C03637=1030.012,334.966,368.080,171.691,46.330,159.041
C03638=1030.005,334.718,368.116,171.685,46.330,159.040
C03639=1029.998,334.472,368.152,171.679,46.328,159.039
C03640=1029.990,334.224,368.188,171.674,46.328,159.038
C03641=1029.982,333.977,368.224,171.668,46.327,159.038
C03642=1029.975,333.730,368.260,171.662,46.326,159.037
C03643=1029.968,333.482,368.296,171.656,46.326,159.036
C03644=1029.961,333.235,368.331,171.652,46.326,159.035
C03645=1029.953,332.988,368.368,171.646,46.325,159.034
C03646=1029.945,332.740,368.403,171.640,46.325,159.034
C03647=1029.938,332.493,368.438,171.635,46.324,159.033
C03648=1029.930,332.246,368.475,171.629,46.323,159.032
C03649=1029.924,331.998,368.510,171.623,46.323,159.031
C03650=1029.916,331.751,368.546,171.617,46.322,159.030
C03651=1029.909,331.504,368.581,171.612,46.321,159.030
C03652=1029.901,331.256,368.617,171.606,46.321,159.029
C03653=1029.895,331.009,368.653,171.601,46.321,159.028
C03654=1029.886,330.762,368.688,171.596,46.320,159.027
C03655=1029.879,330.514,368.723,171.590,46.319,159.027
C03656=1029.872,330.267,368.759,171.584,46.319,159.026
C03657=1029.865,330.019,368.795,171.579,46.319,159.025
C03658=1029.857,329.772,368.831,171.574,46.318,159.024
C03659=1029.851,329.525,368.866,171.569,46.317,159.024
C03660=1029.843,329.277,368.902,171.563,46.317,159.023
C03661=1029.835,329.030,368.937,171.557,46.317,159.022
C03662=1029.829,328.783,368.972,171.552,46.316,159.021
C03663=1029.821,328.535,369.008,171.546,46.315,159.021
C03664=1029.814,328.288,369.043,171.541,46.316,159.020
C03665=1029.807,328.040,369.079,171.536,46.315,159.019
C03666=1029.800,327.793,369.115,171.530,46.314,159.018
C03667=1029.792,327.546,369.149,171.525,46.314,159.018
C03668=1029.785,327.298,369.185,171.519,46.313,159.017
C03669=1029.777,327.051,369.219,171.514,46.313,159.016
C03670=1029.769,326.803,369.254,171.509,46.313,159.015
C03671=1029.762,326.556,369.289,171.503,46.313,159.015
C03672=1029.755,326.309,369.324,171.498,46.313,159.014
C03673=1029.748,326.061,369.359,171.493,46.312,159.013
C03674=1029.740,325.814,369.394,171.487,46.312,159.013
C03675=1029.733,325.566,369.429,171.482,46.311,159.012
C03676=1029.725,325.319,369.464,171.477,46.311,159.011
C03677=1029.718,325.071,369.498,171.471,46.311,159.011
C03678=1029.711,324.824,369.533,171.466,46.310,159.010
C03679=1029.703,324.576,369.568,171.460,46.310,159.009
C03680=1029.696,324.329,369.604,171.456,46.310,159.009
C03681=1029.689,324.081,369.637,171.450,46.310,159.008
C03682=1029.682,323.833,369.673,171.444,46.310,159.007
C03683=1029.674,323.586,369.707,171.440,46.310,159.007
C03684=1029.666,323.339,369.742,171.434,46.310,159.006
C03685=1029.660,323.092,369.777,171.429,46.309,159.005
C03686=1029.652,322.844,369.812,171.424,46.309,159.005
C03687=1029.645,322.596,369.846,171.419,46.309,159.004
C03688=1029.638,322.349,369.881,171.413,46.309,159.003
C03689=1029.630,322.102,369.915,171.408,46.308,159.003
C03690=1029.624,321.891,369.946,171.404,46.308,159.002
C03691=1029.618,321.680,369.974,171.399,46.308,159.002
C03692=1029.612,321.470,370.004,171.395,46.308,159.001
C03693=1029.605,321.259,370.033,171.390,46.308,159.000
C03694=1029.600,321.049,370.063,171.386,46.307,159.000
C03695=1029.593,320.838,370.093,171.381,46.307,158.999
C03696=1029.588,320.627,370.122,171.377,46.307,158.999
C03697=1029.581,320.417,370.151,171.373,46.307,158.998
C03698=1029.575,320.169,370.186,171.367,46.307,158.998
C03699=1029.567,319.922,370.220,171.363,46.306,158.997
C03700=1029.560,319.674,370.255,171.357,46.306,158.996
C03701=1029.553,319.426,370.289,171.352,46.306,158.996
C03702=1029.545,319.179,370.324,171.347,46.306,158.995
C03703=1029.539,318.931,370.358,171.342,46.306,158.994
C03704=1029.531,318.684,370.393,171.337,46.306,158.994
C03705=1029.525,318.436,370.427,171.332,46.306,158.993
C03706=1029.517,318.189,370.462,171.327,46.306,158.993
C03707=1029.510,317.941,370.495,171.322,46.306,158.992
C03708=1029.503,317.694,370.531,171.317,46.305,158.991
C03709=1029.496,317.446,370.564,171.311,46.305,158.991
C03710=1029.489,317.199,370.599,171.307,46.305,158.990
C03711=1029.482,316.951,370.633,171.301,46.305,158.989
C03712=1029.475,316.703,370.667,171.297,46.305,158.989
C03713=1029.468,316.456,370.702,171.291,46.305,158.988
C03714=1029.462,316.209,370.736,171.286,46.305,158.988
C03715=1029.454,315.961,370.770,171.282,46.305,158.987
C03716=1029.448,315.714,370.805,171.276,46.305,158.987
C03717=1029.440,315.466,370.839,171.272,46.305,158.986
C03718=1029.433,315.219,370.872,171.266,46.305,158.985
C03719=1029.427,314.971,370.907,171.262,46.305,158.985
C03720=1029.419,314.724,370.941,171.257,46.305,158.984
C03721=1029.412,314.476,370.975,171.251,46.305,158.984
C03722=1029.406,314.229,371.009,171.247,46.305,158.983
C03723=1029.399,313.981,371.043,171.241,46.305,158.982
C03724=1029.392,313.734,371.078,171.237,46.305,158.982
C03725=1029.385,313.486,371.112,171.232,46.305,158.981
C03726=1029.378,313.238,371.146,171.227,46.305,158.981
C03727=1029.371,312.991,371.180,171.222,46.305,158.980
C03728=1029.365,312.743,371.214,171.218,46.305,158.980
C03729=1029.358,312.496,371.248,171.212,46.305,158.979
C03730=1029.351,312.248,371.282,171.207,46.305,158.978
C03731=1029.344,312.000,371.316,171.203,46.305,158.978
C03732=1029.337,311.753,371.349,171.197,46.305,158.977
C03733=1029.331,311.505,371.384,171.193,46.305,158.977
C03734=1029.324,311.257,371.417,171.188,46.305,158.976
C03735=1029.317,311.010,371.451,171.183,46.306,158.976
C03736=1029.310,310.763,371.485,171.178,46.305,158.975
C03737=1029.303,310.515,371.519,171.174,46.306,158.975
C03738=1029.295,310.268,371.552,171.168,46.306,158.974
C03739=1029.288,310.019,371.585,171.164,46.306,158.974
C03740=1029.281,309.772,371.618,171.158,46.306,158.973
C03741=1029.273,309.525,371.652,171.154,46.307,158.973
C03742=1029.266,309.277,371.685,171.149,46.306,158.972
C03743=1029.259,309.029,371.719,171.144,46.307,158.972
C03744=1029.253,308.782,371.752,171.140,46.307,158.971
C03745=1029.245,308.535,371.785,171.134,46.307,158.970
C03746=1029.238,308.286,371.818,171.130,46.308,158.970
C03747=1029.231,308.040,371.852,171.126,46.308,158.970
C03748=1029.224,307.791,371.885,171.120,46.308,158.969
C03749=1029.216,307.544,371.918,171.116,46.309,158.969
C03750=1029.205,307.127,371.974,171.108,46.309,158.968
C03751=1029.193,306.711,372.030,171.099,46.309,158.967
C03752=1029.181,306.295,372.086,171.091,46.310,158.966
C03753=1029.170,305.879,372.141,171.084,46.311,158.965
C03754=1029.162,305.631,372.175,171.079,46.311,158.965
C03755=1029.155,305.384,372.207,171.074,46.312,158.964
C03756=1029.148,305.136,372.241,171.069,46.311,158.964
C03757=1029.141,304.888,372.274,171.065,46.312,158.963
C03758=1029.134,304.640,372.306,171.060,46.312,158.963
C03759=1029.127,304.393,372.340,171.055,46.313,158.963
C03760=1029.121,304.145,372.373,171.051,46.313,158.962
C03761=1029.113,303.897,372.405,171.046,46.313,158.961
C03762=1029.107,303.650,372.439,171.041,46.314,158.961
C03763=1029.100,303.402,372.472,171.037,46.314,158.961
C03764=1029.093,303.154,372.505,171.033,46.314,158.960
C03765=1029.085,302.907,372.538,171.027,46.315,158.960
C03766=1029.079,302.659,372.571,171.023,46.316,158.959
C03767=1029.072,302.411,372.604,171.019,46.316,158.959
C03768=1029.065,302.164,372.636,171.014,46.316,158.958
C03769=1029.058,301.916,372.670,171.009,46.316,158.958
C03770=1029.052,301.668,372.702,171.004,46.317,158.957
C03771=1029.044,301.420,372.735,171.000,46.317,158.957
C03772=1029.038,301.173,372.768,170.996,46.318,158.957
C03773=1029.031,300.925,372.801,170.990,46.318,158.956
C03774=1029.025,300.677,372.834,170.986,46.319,158.956
C03775=1029.017,300.430,372.867,170.982,46.319,158.955
C03776=1029.010,300.182,372.900,170.977,46.319,158.955
C03777=1029.004,299.934,372.932,170.973,46.320,158.954
C03778=1028.996,299.686,372.965,170.968,46.320,158.954
C03779=1028.990,299.439,372.998,170.963,46.321,158.954
C03780=1028.983,299.191,373.031,170.959,46.321,158.953
C03781=1028.976,298.943,373.063,170.955,46.322,158.953
C03782=1028.970,298.696,373.096,170.950,46.322,158.952
C03783=1028.963,298.447,373.129,170.945,46.323,158.952
C03784=1028.956,298.200,373.161,170.941,46.323,158.951
C03785=1028.950,297.953,373.194,170.936,46.323,158.951
C03786=1028.943,297.704,373.227,170.932,46.324,158.951
C03787=1028.936,297.457,373.259,170.928,46.324,158.950
C03788=1028.930,297.209,373.292,170.922,46.325,158.950
C03789=1028.923,296.962,373.324,170.918,46.325,158.949
C03790=1028.916,296.714,373.357,170.914,46.326,158.949
C03791=1028.909,296.466,373.390,170.909,46.326,158.948
C03792=1028.903,296.219,373.422,170.905,46.327,158.948
C03793=1028.896,295.970,373.454,170.901,46.328,158.948
C03794=1028.889,295.722,373.487,170.897,46.328,158.947
C03795=1028.883,295.475,373.520,170.891,46.329,158.947
C03796=1028.876,295.228,373.552,170.887,46.329,158.946
C03797=1028.870,294.980,373.584,170.883,46.329,158.946
C03798=1028.863,294.732,373.618,170.878,46.330,158.946
C03799=1028.856,294.484,373.649,170.874,46.331,158.945
C03800=1028.850,294.236,373.682,170.870,46.331,158.945
C03801=1028.843,293.989,373.714,170.866,46.332,158.945
C03802=1028.836,293.740,373.746,170.860,46.332,158.944
C03803=1028.829,293.493,373.778,170.856,46.333,158.944
C03804=1028.822,293.245,373.811,170.852,46.334,158.943
C03805=1028.816,292.997,373.843,170.848,46.334,158.943
C03806=1028.804,292.598,373.894,170.840,46.335,158.942
C03807=1028.794,292.199,373.946,170.834,46.336,158.942
C03808=1028.783,291.800,373.998,170.827,46.337,158.941
C03809=1028.772,291.400,374.049,170.820,46.339,158.941
C03810=1028.765,291.153,374.081,170.815,46.339,158.940
C03811=1028.759,290.905,374.113,170.811,46.340,158.940
C03812=1028.752,290.657,374.145,170.807,46.341,158.940
C03813=1028.745,290.409,374.176,170.803,46.341,158.939
C03814=1028.738,290.161,374.208,170.799,46.342,158.939
C03815=1028.731,289.914,374.240,170.793,46.343,158.939
C03816=1028.725,289.665,374.272,170.789,46.344,158.938
C03817=1028.718,289.417,374.304,170.785,46.344,158.938
C03818=1028.711,289.170,374.336,170.781,46.345,158.938
C03819=1028.704,288.922,374.367,170.777,46.346,158.938
C03820=1028.697,288.674,374.399,170.772,46.347,158.937
C03821=1028.690,288.427,374.431,170.768,46.348,158.937
C03822=1028.684,288.179,374.463,170.764,46.348,158.936
C03823=1028.677,287.930,374.495,170.759,46.350,158.936
C03824=1028.670,287.682,374.526,170.755,46.350,158.936
C03825=1028.664,287.434,374.558,170.751,46.351,158.935
C03826=1028.657,287.187,374.590,170.747,46.352,158.935
C03827=1028.650,286.939,374.621,170.742,46.352,158.935
C03828=1028.643,286.691,374.653,170.738,46.353,158.935
C03829=1028.636,286.443,374.684,170.734,46.354,158.934
C03830=1028.630,286.196,374.716,170.730,46.355,158.934
C03831=1028.624,285.947,374.748,170.726,46.356,158.934
C03832=1028.617,285.699,374.779,170.722,46.357,158.933
C03833=1028.609,285.452,374.810,170.717,46.357,158.933
C03834=1028.603,285.204,374.841,170.712,46.359,158.933
C03835=1028.596,284.956,374.873,170.708,46.360,158.932
C03836=1028.589,284.708,374.904,170.704,46.361,158.932
C03837=1028.583,284.460,374.936,170.700,46.361,158.932
C03838=1028.576,284.212,374.967,170.696,46.362,158.932
C03839=1028.569,283.964,374.999,170.692,46.363,158.931
C03840=1028.562,283.716,375.030,170.688,46.364,158.931
C03841=1028.556,283.469,375.061,170.684,46.365,158.931
C03842=1028.548,283.221,375.092,170.680,46.366,158.931
C03843=1028.542,282.973,375.124,170.676,46.367,158.930
C03844=1028.535,282.725,375.154,170.671,46.368,158.930
C03845=1028.528,282.477,375.186,170.667,46.369,158.930
C03846=1028.522,282.229,375.217,170.663,46.370,158.929
C03847=1028.515,281.981,375.249,170.658,46.371,158.929
C03848=1028.508,281.733,375.280,170.654,46.372,158.929
C03849=1028.501,281.485,375.312,170.650,46.373,158.929
C03850=1028.495,281.237,375.342,170.646,46.373,158.928
C03851=1028.488,280.989,375.373,170.642,46.374,158.928
C03852=1028.481,280.741,375.405,170.638,46.375,158.928
C03853=1028.475,280.494,375.436,170.634,46.376,158.927
C03854=1028.468,280.245,375.466,170.630,46.377,158.927
C03855=1028.462,279.997,375.498,170.626,46.378,158.927
C03856=1028.455,279.749,375.529,170.622,46.379,158.927
C03857=1028.448,279.501,375.560,170.618,46.381,158.926
C03858=1028.442,279.253,375.591,170.614,46.382,158.926
C03859=1028.434,279.005,375.622,170.610,46.383,158.926
C03860=1028.428,278.758,375.653,170.606,46.384,158.926
C03861=1028.422,278.510,375.684,170.601,46.385,158.925
C03862=1028.411,278.122,375.733,170.595,46.386,158.925
C03863=1028.401,277.736,375.781,170.589,46.388,158.925
C03864=1028.391,277.349,375.829,170.582,46.389,158.924
C03865=1028.380,276.962,375.878,170.576,46.391,158.924
C03866=1028.373,276.713,375.908,170.572,46.392,158.924
C03867=1028.367,276.466,375.938,170.568,46.393,158.923
C03868=1028.360,276.218,375.969,170.564,46.394,158.923
C03869=1028.354,275.969,376.000,170.560,46.396,158.923
C03870=1028.346,275.722,376.031,170.556,46.397,158.923
C03871=1028.340,275.474,376.061,170.552,46.398,158.923
C03872=1028.333,275.226,376.092,170.548,46.399,158.922
C03873=1028.327,274.978,376.123,170.544,46.400,158.922
C03874=1028.320,274.729,376.154,170.540,46.401,158.922
C03875=1028.313,274.482,376.185,170.536,46.403,158.922
C03876=1028.307,274.234,376.215,170.532,46.404,158.922
C03877=1028.300,273.985,376.246,170.528,46.405,158.921
C03878=1028.293,273.737,376.276,170.524,46.406,158.921
C03879=1028.287,273.490,376.307,170.520,46.407,158.921
C03880=1028.280,273.242,376.337,170.516,46.408,158.921
C03881=1028.274,272.993,376.368,170.512,46.409,158.921
C03882=1028.266,272.745,376.398,170.508,46.410,158.920
C03883=1028.260,272.498,376.429,170.504,46.411,158.920
C03884=1028.254,272.249,376.460,170.501,46.413,158.920
C03885=1028.247,272.001,376.490,170.497,46.414,158.920
C03886=1028.241,271.753,376.520,170.493,46.415,158.919
C03887=1028.234,271.505,376.550,170.489,46.417,158.919
C03888=1028.227,271.257,376.582,170.485,46.418,158.919
C03889=1028.220,271.009,376.611,170.481,46.419,158.919
C03890=1028.214,270.761,376.642,170.477,46.421,158.919
C03891=1028.207,270.513,376.672,170.474,46.421,158.919
C03892=1028.201,270.265,376.702,170.470,46.422,158.918
C03893=1028.194,270.017,376.733,170.466,46.424,158.918
C03894=1028.187,269.768,376.763,170.462,46.425,158.918
C03895=1028.181,269.521,376.793,170.458,46.427,158.918
C03896=1028.174,269.272,376.823,170.454,46.428,158.918
C03897=1028.167,269.024,376.854,170.450,46.429,158.917
C03898=1028.161,268.776,376.884,170.446,46.430,158.917
C03899=1028.154,268.528,376.914,170.442,46.431,158.917
C03900=1028.148,268.280,376.944,170.439,46.433,158.917
C03901=1028.141,268.032,376.974,170.435,46.434,158.917
C03902=1028.133,267.784,377.004,170.431,46.436,158.917
C03903=1028.128,267.536,377.035,170.427,46.437,158.916
C03904=1028.121,267.288,377.065,170.423,46.438,158.916
C03905=1028.114,267.040,377.095,170.419,46.440,158.916
C03906=1028.108,266.791,377.125,170.415,46.441,158.916
C03907=1028.101,266.544,377.154,170.411,46.442,158.916
C03908=1028.094,266.296,377.184,170.407,46.444,158.916
C03909=1028.088,266.047,377.215,170.403,46.445,158.916
C03910=1028.081,265.799,377.245,170.401,46.446,158.916
C03911=1028.074,265.551,377.274,170.397,46.447,158.915
C03912=1028.068,265.303,377.304,170.393,46.449,158.915
C03913=1028.061,265.055,377.335,170.389,46.451,158.915
C03914=1028.055,264.807,377.365,170.385,46.452,158.915
C03915=1028.048,264.558,377.394,170.381,46.453,158.915
C03916=1028.041,264.311,377.424,170.377,46.454,158.915
C03917=1028.034,264.063,377.454,170.374,46.456,158.914
C03918=1028.024,263.680,377.500,170.368,46.458,158.914
C03919=1028.014,263.298,377.546,170.362,46.460,158.914
C03920=1028.004,262.915,377.592,170.356,46.463,158.914
C03921=1027.994,262.533,377.637,170.350,46.465,158.914
C03922=1027.987,262.285,377.668,170.347,46.466,158.914
C03923=1027.981,262.037,377.697,170.343,46.467,158.913
C03924=1027.974,261.788,377.727,170.339,46.469,158.913
C03925=1027.968,261.540,377.756,170.335,46.471,158.913
C03926=1027.961,261.293,377.786,170.331,46.472,158.913
C03927=1027.954,261.044,377.816,170.328,46.473,158.913
C03928=1027.948,260.796,377.845,170.325,46.475,158.913
C03929=1027.941,260.548,377.874,170.321,46.477,158.913
C03930=1027.934,260.300,377.904,170.317,46.478,158.913
C03931=1027.927,260.051,377.934,170.313,46.480,158.913
C03932=1027.921,259.804,377.963,170.310,46.482,158.912
C03933=1027.913,259.555,377.992,170.306,46.483,158.912
C03934=1027.907,259.307,378.021,170.302,46.484,158.912
C03935=1027.900,259.059,378.051,170.298,46.486,158.912
C03936=1027.894,258.811,378.080,170.294,46.488,158.912
C03937=1027.887,258.563,378.109,170.291,46.489,158.912
C03938=1027.880,258.314,378.138,170.287,46.491,158.912
C03939=1027.873,258.067,378.168,170.283,46.493,158.912
C03940=1027.866,257.818,378.197,170.279,46.494,158.912
C03941=1027.860,257.570,378.226,170.277,46.496,158.912
C03942=1027.853,257.321,378.256,170.273,46.497,158.912
C03943=1027.846,257.074,378.285,170.269,46.499,158.912
C03944=1027.840,256.825,378.314,170.265,46.501,158.911
C03945=1027.833,256.577,378.343,170.262,46.502,158.911
C03946=1027.827,256.328,378.373,170.258,46.504,158.911
C03947=1027.820,256.081,378.401,170.254,46.506,158.911
C03948=1027.812,255.832,378.431,170.250,46.507,158.911
C03949=1027.806,255.584,378.460,170.247,46.509,158.911
C03950=1027.799,255.335,378.490,170.243,46.511,158.911
C03951=1027.793,255.087,378.519,170.240,46.512,158.911
C03952=1027.786,254.839,378.547,170.236,46.514,158.911
C03953=1027.779,254.591,378.576,170.233,46.516,158.911
C03954=1027.773,254.342,378.605,170.229,46.517,158.911
C03955=1027.767,254.094,378.635,170.225,46.519,158.911
C03956=1027.760,253.847,378.663,170.221,46.521,158.911
C03957=1027.753,253.598,378.693,170.217,46.522,158.910
C03958=1027.746,253.350,378.722,170.214,46.524,158.910
C03959=1027.740,253.102,378.751,170.211,46.525,158.910
C03960=1027.733,252.853,378.781,170.207,46.527,158.910
C03961=1027.726,252.605,378.809,170.203,46.529,158.910
C03962=1027.720,252.357,378.838,170.200,46.530,158.910
C03963=1027.714,252.109,378.867,170.196,46.532,158.910
C03964=1027.707,251.860,378.897,170.192,46.534,158.910
C03965=1027.700,251.612,378.925,170.188,46.535,158.910
C03966=1027.694,251.364,378.954,170.186,46.537,158.910
C03967=1027.687,251.116,378.983,170.182,46.539,158.910
C03968=1027.681,250.867,379.012,170.179,46.541,158.910
C03969=1027.674,250.620,379.041,170.175,46.542,158.910
C03970=1027.668,250.371,379.069,170.171,46.544,158.910
C03971=1027.661,250.123,379.098,170.167,46.546,158.910
C03972=1027.655,249.875,379.127,170.164,46.547,158.910
C03973=1027.648,249.626,379.156,170.161,46.549,158.909
C03974=1027.638,249.242,379.201,170.155,46.552,158.909
C03975=1027.628,248.859,379.246,170.150,46.555,158.909
C03976=1027.618,248.475,379.290,170.144,46.557,158.909
C03977=1027.608,248.091,379.335,170.139,46.560,158.909
C03978=1027.601,247.843,379.364,170.135,46.562,158.909
C03979=1027.595,247.594,379.392,170.132,46.563,158.909
C03980=1027.589,247.346,379.421,170.129,46.565,158.909
C03981=1027.583,247.098,379.450,170.125,46.567,158.909
C03982=1027.576,246.850,379.478,170.121,46.569,158.909
C03983=1027.569,246.601,379.508,170.118,46.571,158.909
C03984=1027.563,246.353,379.536,170.115,46.572,158.909
C03985=1027.557,246.105,379.565,170.111,46.574,158.909
C03986=1027.550,245.857,379.594,170.107,46.575,158.909
C03987=1027.543,245.609,379.623,170.104,46.578,158.909
C03988=1027.537,245.360,379.651,170.101,46.579,158.909
C03989=1027.531,245.112,379.680,170.097,46.581,158.909
C03990=1027.524,244.864,379.709,170.094,46.583,158.909
C03991=1027.518,244.615,379.737,170.090,46.585,158.909
C03992=1027.512,244.367,379.766,170.086,46.587,158.909
C03993=1027.505,244.119,379.794,170.084,46.588,158.909
C03994=1027.499,243.870,379.823,170.080,46.590,158.909
C03995=1027.492,243.623,379.851,170.076,46.592,158.909
C03996=1027.486,243.374,379.879,170.073,46.594,158.909
C03997=1027.479,243.125,379.908,170.069,46.596,158.909
C03998=1027.473,242.877,379.937,170.066,46.597,158.909
C03999=1027.466,242.629,379.965,170.063,46.599,158.909
C04000=1027.460,242.380,379.993,170.059,46.601,158.909
C04001=1027.453,242.132,380.022,170.055,46.603,158.909
C04002=1027.447,241.883,380.050,170.053,46.605,158.909
C04003=1027.440,241.636,380.079,170.049,46.607,158.909
C04004=1027.434,241.387,380.107,170.046,46.609,158.909
C04005=1027.427,241.139,380.135,170.042,46.611,158.909
C04006=1027.420,240.891,380.163,170.038,46.613,158.909
C04007=1027.414,240.642,380.192,170.036,46.615,158.909
C04008=1027.407,240.394,380.220,170.032,46.616,158.909
C04009=1027.401,240.145,380.248,170.029,46.619,158.909
C04010=1027.394,239.897,380.277,170.025,46.620,158.909
C04011=1027.388,239.649,380.304,170.021,46.623,158.909
C04012=1027.382,239.400,380.333,170.019,46.624,158.909
C04013=1027.375,239.152,380.361,170.015,46.626,158.909
C04014=1027.368,238.904,380.389,170.011,46.628,158.909
C04015=1027.361,238.656,380.417,170.008,46.630,158.909
C04016=1027.355,238.407,380.444,170.005,46.633,158.909
C04017=1027.348,238.159,380.473,170.002,46.634,158.909
C04018=1027.342,237.911,380.501,169.998,46.636,158.909
C04019=1027.335,237.662,380.529,169.995,46.638,158.909
C04020=1027.328,237.414,380.557,169.991,46.641,158.909
C04021=1027.322,237.165,380.584,169.988,46.643,158.909
C04022=1027.315,236.917,380.613,169.985,46.644,158.909
C04023=1027.309,236.669,380.641,169.981,46.647,158.909
C04024=1027.302,236.420,380.669,169.978,46.649,158.909
C04025=1027.295,236.172,380.696,169.974,46.651,158.909
C04026=1027.289,235.924,380.724,169.971,46.653,158.909
C04027=1027.283,235.676,380.752,169.968,46.655,158.909
C04028=1027.276,235.427,380.779,169.965,46.657,158.909
C04029=1027.270,235.178,380.808,169.961,46.659,158.909
C04030=1027.259,234.789,380.851,169.956,46.663,158.909
C04031=1027.249,234.398,380.896,169.950,46.665,158.909
C04032=1027.239,234.009,380.939,169.945,46.669,158.910
C04033=1027.229,233.619,380.982,169.940,46.672,158.910
C04034=1027.222,233.370,381.010,169.937,46.674,158.910
C04035=1027.215,233.122,381.038,169.934,46.676,158.910
C04036=1027.209,232.873,381.066,169.930,46.678,158.910
C04037=1027.202,232.625,381.093,169.927,46.681,158.910
C04038=1027.196,232.377,381.121,169.924,46.682,158.910
C04039=1027.189,232.129,381.148,169.921,46.685,158.910
C04040=1027.183,231.880,381.176,169.917,46.687,158.910
C04041=1027.177,231.631,381.205,169.914,46.689,158.910
C04042=1027.170,231.383,381.232,169.911,46.691,158.910
C04043=1027.163,231.135,381.260,169.908,46.693,158.910
C04044=1027.157,230.887,381.287,169.904,46.695,158.910
C04045=1027.150,230.638,381.315,169.901,46.698,158.910
C04046=1027.144,230.390,381.343,169.898,46.700,158.911
C04047=1027.137,230.141,381.370,169.894,46.701,158.910
C04048=1027.131,229.892,381.398,169.891,46.704,158.911
C04049=1027.124,229.644,381.425,169.888,46.706,158.911
C04050=1027.118,229.396,381.453,169.885,46.708,158.911
C04051=1027.111,229.148,381.480,169.882,46.711,158.911
C04052=1027.105,228.899,381.508,169.878,46.713,158.911
C04053=1027.098,228.650,381.535,169.875,46.715,158.911
C04054=1027.092,228.402,381.563,169.872,46.717,158.911
C04055=1027.085,228.154,381.590,169.869,46.719,158.911
C04056=1027.079,227.906,381.618,169.865,46.721,158.911
C04057=1027.072,227.657,381.644,169.862,46.724,158.911
C04058=1027.065,227.408,381.672,169.859,46.726,158.911
C04059=1027.059,227.161,381.699,169.856,46.728,158.911
C04060=1027.053,226.912,381.726,169.852,46.730,158.912
C04061=1027.046,226.663,381.754,169.849,46.733,158.912
C04062=1027.038,226.415,381.781,169.846,46.735,158.912
C04063=1027.033,226.167,381.808,169.843,46.737,158.912
C04064=1027.026,225.918,381.836,169.839,46.740,158.912
C04065=1027.020,225.669,381.863,169.836,46.742,158.912
C04066=1027.012,225.421,381.890,169.832,46.744,158.912
C04067=1027.006,225.173,381.918,169.830,46.746,158.912
C04068=1027.000,224.924,381.944,169.827,46.749,158.912
C04069=1026.992,224.676,381.971,169.823,46.751,158.912
C04070=1026.986,224.427,381.998,169.820,46.753,158.912
C04071=1026.980,224.179,382.026,169.817,46.755,158.913
C04072=1026.974,223.930,382.053,169.814,46.758,158.913
C04073=1026.966,223.682,382.080,169.811,46.761,158.913
C04074=1026.960,223.433,382.107,169.807,46.763,158.913
C04075=1026.954,223.185,382.134,169.805,46.765,158.913
C04076=1026.947,222.937,382.161,169.801,46.768,158.913
C04077=1026.940,222.688,382.188,169.798,46.770,158.913
C04078=1026.934,222.440,382.215,169.794,46.772,158.913
C04079=1026.927,222.191,382.243,169.792,46.774,158.914
C04080=1026.920,221.943,382.269,169.788,46.777,158.914
C04081=1026.914,221.695,382.297,169.785,46.779,158.914
C04082=1026.908,221.446,382.324,169.782,46.781,158.914
C04083=1026.901,221.197,382.350,169.779,46.784,158.914
C04084=1026.895,220.949,382.377,169.776,46.786,158.914
C04085=1026.888,220.700,382.404,169.772,46.789,158.914
C04086=1026.877,220.303,382.448,169.767,46.792,158.914
C04087=1026.868,219.905,382.491,169.762,46.796,158.915
C04088=1026.857,219.508,382.534,169.758,46.800,158.915
C04089=1026.847,219.110,382.577,169.753,46.803,158.915
C04090=1026.840,218.861,382.604,169.750,46.806,158.915
C04091=1026.833,218.613,382.631,169.746,46.809,158.915
C04092=1026.826,218.365,382.657,169.743,46.811,158.915
C04093=1026.820,218.116,382.684,169.741,46.814,158.916
C04094=1026.813,217.868,382.711,169.737,46.816,158.916
C04095=1026.807,217.619,382.738,169.734,46.818,158.916
C04096=1026.800,217.370,382.764,169.730,46.821,158.916
C04097=1026.794,217.122,382.791,169.728,46.823,158.916
C04098=1026.787,216.873,382.817,169.725,46.826,158.916
C04099=1026.780,216.625,382.843,169.721,46.828,158.916
C04100=1026.774,216.377,382.871,169.718,46.831,158.917
C04101=1026.767,216.128,382.897,169.716,46.833,158.917
C04102=1026.761,215.880,382.924,169.712,46.836,158.917
C04103=1026.754,215.631,382.950,169.709,46.839,158.917
C04104=1026.748,215.382,382.977,169.706,46.841,158.917
C04105=1026.741,215.134,383.004,169.703,46.843,158.917
C04106=1026.734,214.886,383.030,169.700,46.846,158.918
C04107=1026.728,214.637,383.057,169.697,46.848,158.918
C04108=1026.721,214.388,383.083,169.693,46.851,158.918
C04109=1026.715,214.140,383.110,169.691,46.853,158.918
C04110=1026.708,213.891,383.137,169.687,46.856,158.918
C04111=1026.701,213.643,383.163,169.684,46.859,158.918
C04112=1026.695,213.394,383.190,169.682,46.861,158.919
C04113=1026.688,213.146,383.216,169.678,46.863,158.919
C04114=1026.682,212.897,383.243,169.675,46.866,158.919
C04115=1026.675,212.649,383.269,169.672,46.869,158.919
C04116=1026.669,212.400,383.296,169.669,46.871,158.919
C04117=1026.662,212.152,383.322,169.666,46.874,158.919
C04118=1026.655,211.903,383.348,169.663,46.876,158.919
C04119=1026.650,211.655,383.375,169.661,46.879,158.920
C04120=1026.642,211.406,383.402,169.657,46.881,158.920
C04121=1026.637,211.158,383.428,169.654,46.884,158.920
C04122=1026.630,210.909,383.455,169.651,46.886,158.920
C04123=1026.623,210.661,383.481,169.648,46.889,158.920
C04124=1026.617,210.412,383.508,169.645,46.892,158.921
C04125=1026.610,210.163,383.533,169.641,46.894,158.921
C04126=1026.604,209.915,383.559,169.639,46.897,158.921
C04127=1026.597,209.666,383.585,169.636,46.899,158.921
C04128=1026.590,209.418,383.612,169.633,46.902,158.921
C04129=1026.584,209.169,383.639,169.629,46.905,158.921
C04130=1026.577,208.921,383.665,169.627,46.907,158.922
C04131=1026.570,208.673,383.691,169.624,46.910,158.922
C04132=1026.564,208.424,383.716,169.620,46.913,158.922
C04133=1026.558,208.175,383.743,169.618,46.915,158.922
C04134=1026.551,207.927,383.769,169.615,46.918,158.922
C04135=1026.544,207.678,383.796,169.612,46.921,158.923
C04136=1026.538,207.429,383.821,169.608,46.923,158.923
C04137=1026.531,207.181,383.847,169.606,46.926,158.923
C04138=1026.524,206.933,383.874,169.603,46.928,158.923
C04139=1026.518,206.685,383.900,169.599,46.931,158.923
C04140=1026.512,206.435,383.926,169.597,46.934,158.924
C04141=1026.505,206.187,383.952,169.594,46.936,158.924
C04142=1026.494,205.793,383.994,169.589,46.941,158.924
C04143=1026.484,205.399,384.034,169.584,46.945,158.924
C04144=1026.474,205.006,384.076,169.580,46.950,158.925
C04145=1026.463,204.611,384.116,169.575,46.954,158.925
C04146=1026.439,203.573,384.219,169.186,46.851,158.855
C04147=1026.432,203.324,384.244,169.182,46.855,158.856
C04148=1026.427,203.076,384.268,169.178,46.858,158.856
C04149=1026.421,202.827,384.292,169.174,46.862,158.856
C04150=1026.415,202.578,384.317,169.170,46.865,158.856
C04151=1026.409,202.329,384.342,169.166,46.869,158.857
C04152=1026.403,202.081,384.366,169.162,46.873,158.857
C04153=1026.397,201.832,384.390,169.158,46.876,158.857
C04154=1026.392,201.583,384.415,169.155,46.880,158.857
C04155=1026.386,201.334,384.439,169.151,46.883,158.858
C04156=1026.381,201.086,384.464,169.147,46.887,158.858
C04157=1026.375,200.838,384.488,169.143,46.890,158.858
C04158=1026.369,200.588,384.512,169.139,46.894,158.858
C04159=1026.363,200.340,384.537,169.135,46.897,158.859
C04160=1026.357,200.090,384.561,169.131,46.901,158.859
C04161=1026.351,199.842,384.585,169.127,46.904,158.859
C04162=1026.345,199.593,384.610,169.124,46.908,158.859
C04163=1026.339,199.345,384.633,169.119,46.912,158.860
C04164=1026.334,199.095,384.658,169.116,46.915,158.860
C04165=1026.328,198.847,384.682,169.112,46.919,158.860
C04166=1026.321,198.598,384.706,169.107,46.923,158.860
C04167=1026.316,198.350,384.730,169.104,46.927,158.861
C04168=1026.309,198.101,384.754,169.100,46.931,158.861
C04169=1026.304,197.851,384.777,169.095,46.934,158.861
C04170=1026.298,197.603,384.801,169.092,46.938,158.862
C04171=1026.292,197.354,384.826,169.089,46.942,158.862
C04172=1026.286,197.105,384.849,169.084,46.945,158.862
C04173=1026.279,196.856,384.873,169.081,46.949,158.862
C04174=1026.274,196.608,384.898,169.077,46.953,158.863
C04175=1026.268,196.360,384.921,169.072,46.956,158.863
C04176=1026.262,196.110,384.945,169.069,46.960,158.863
C04177=1026.256,195.861,384.969,169.065,46.964,158.864
C04178=1026.251,195.613,384.993,169.062,46.967,158.864
C04179=1026.244,195.364,385.017,169.058,46.971,158.864
C04180=1026.238,195.116,385.041,169.054,46.975,158.864
C04181=1026.233,194.866,385.064,169.050,46.978,158.865
C04182=1026.227,194.617,385.088,169.046,46.982,158.865
C04183=1026.221,194.369,385.113,169.042,46.986,158.865
C04184=1026.215,194.121,385.136,169.039,46.989,158.865
C04185=1026.209,193.871,385.160,169.035,46.993,158.866
C04186=1026.204,193.622,385.184,169.031,46.997,158.866
C04187=1026.198,193.374,385.208,169.027,47.000,158.866
C04188=1026.192,193.124,385.231,169.023,47.004,158.867
C04189=1026.186,192.876,385.255,169.019,47.008,158.867
C04190=1026.181,192.627,385.279,169.016,47.012,158.867
C04191=1026.175,192.379,385.303,169.012,47.015,158.867
C04192=1026.168,192.129,385.326,169.008,47.019,158.868
C04193=1026.163,191.881,385.351,169.004,47.023,158.868
C04194=1026.157,191.632,385.374,169.001,47.026,158.868
C04195=1026.152,191.383,385.398,168.997,47.030,158.869
C04196=1026.145,191.134,385.422,168.993,47.034,158.869
C04197=1026.140,190.885,385.445,168.989,47.038,158.869
C04198=1026.134,190.637,385.469,168.986,47.041,158.870
C04199=1026.129,190.388,385.492,168.982,47.045,158.870
C04200=1026.123,190.139,385.517,168.978,47.049,158.870
C04201=1026.117,189.890,385.540,168.974,47.053,158.871
C04202=1026.111,189.642,385.563,168.971,47.056,158.871
C04203=1026.106,189.393,385.587,168.967,47.060,158.871
C04204=1026.100,189.144,385.610,168.963,47.064,158.871
C04205=1026.094,188.895,385.635,168.960,47.068,158.872
C04206=1026.088,188.646,385.658,168.956,47.071,158.872
C04207=1026.083,188.410,385.681,168.952,47.075,158.872
C04208=1026.078,188.174,385.703,168.949,47.078,158.872
C04209=1026.072,187.938,385.725,168.945,47.082,158.873
C04210=1026.066,187.702,385.747,168.943,47.086,158.873
C04211=1026.061,187.466,385.770,168.938,47.089,158.873
C04212=1026.056,187.231,385.792,168.935,47.093,158.874
C04213=1026.051,186.994,385.815,168.931,47.096,158.874
C04214=1026.046,186.758,385.837,168.928,47.100,158.874
C04215=1026.040,186.509,385.860,168.925,47.104,158.875
C04216=1026.034,186.260,385.883,168.921,47.107,158.875
C04217=1026.028,186.011,385.908,168.917,47.111,158.875
C04218=1026.022,185.762,385.931,168.914,47.115,158.875
C04219=1026.017,185.514,385.955,168.911,47.118,158.876
C04220=1026.011,185.265,385.978,168.907,47.122,158.876
C04221=1026.006,185.016,386.001,168.903,47.126,158.876
C04222=1026.000,184.767,386.025,168.900,47.129,158.877
C04223=1025.995,184.518,386.048,168.896,47.133,158.877
C04224=1025.989,184.269,386.071,168.892,47.137,158.877
C04225=1025.984,184.021,386.095,168.889,47.140,158.878
C04226=1025.978,183.772,386.118,168.885,47.144,158.878
C04227=1025.973,183.523,386.142,168.881,47.148,158.878
C04228=1025.967,183.274,386.165,168.878,47.152,158.879
C04229=1025.961,183.026,386.188,168.874,47.155,158.879
C04230=1025.956,182.776,386.212,168.871,47.159,158.879
C04231=1025.950,182.527,386.235,168.867,47.163,158.879
C04232=1025.944,182.278,386.258,168.863,47.167,158.880
C04233=1025.938,182.029,386.281,168.860,47.171,158.880
C04234=1025.932,181.781,386.304,168.857,47.175,158.881
C04235=1025.926,181.532,386.327,168.853,47.179,158.881
C04236=1025.920,181.283,386.350,168.849,47.183,158.881
C04237=1025.914,181.035,386.372,168.845,47.187,158.882
C04238=1025.908,180.785,386.395,168.842,47.191,158.882
C04239=1025.902,180.536,386.418,168.839,47.195,158.882
C04240=1025.897,180.287,386.441,168.835,47.199,158.883
C04241=1025.890,180.039,386.463,168.832,47.203,158.883
C04242=1025.885,179.790,386.486,168.828,47.207,158.883
C04243=1025.877,179.481,386.515,168.823,47.212,158.884
C04244=1025.870,179.173,386.543,168.819,47.217,158.884
C04245=1025.862,178.865,386.571,168.815,47.222,158.885
C04246=1025.855,178.556,386.599,168.811,47.227,158.885
C04247=1025.849,178.308,386.622,168.807,47.231,158.886
C04248=1025.844,178.059,386.645,168.803,47.235,158.886
C04249=1025.837,177.810,386.667,168.800,47.239,158.886
C04250=1025.832,177.561,386.689,168.796,47.243,158.887
C04251=1025.826,177.312,386.712,168.793,47.247,158.887
C04252=1025.820,177.063,386.735,168.790,47.250,158.887
C04253=1025.814,176.814,386.758,168.786,47.255,158.888
C04254=1025.808,176.565,386.781,168.782,47.259,158.888
C04255=1025.802,176.316,386.804,168.779,47.263,158.888
C04256=1025.797,176.067,386.826,168.776,47.267,158.889
C04257=1025.791,175.818,386.848,168.772,47.271,158.889
C04258=1025.785,175.569,386.871,168.769,47.275,158.890
C04259=1025.779,175.320,386.894,168.765,47.279,158.890
C04260=1025.773,175.072,386.916,168.761,47.283,158.890
C04261=1025.767,174.822,386.939,168.758,47.287,158.891
C04262=1025.761,174.573,386.962,168.755,47.291,158.891
C04263=1025.756,174.325,386.984,168.752,47.295,158.891
C04264=1025.750,174.076,387.006,168.748,47.299,158.892
C04265=1025.744,173.827,387.029,168.744,47.303,158.892
C04266=1025.739,173.578,387.052,168.741,47.306,158.892
C04267=1025.733,173.329,387.075,168.737,47.310,158.893
C04268=1025.727,173.080,387.096,168.734,47.315,158.893
C04269=1025.721,172.831,387.119,168.731,47.319,158.894
C04270=1025.715,172.582,387.142,168.727,47.323,158.894
C04271=1025.709,172.299,387.167,168.723,47.328,158.894
C04272=1025.702,172.017,387.193,168.720,47.332,158.895
C04273=1025.696,171.733,387.219,168.716,47.336,158.895
C04274=1025.689,171.450,387.244,168.711,47.341,158.896
C04275=1025.684,171.201,387.267,168.709,47.345,158.896
C04276=1025.678,170.952,387.288,168.705,47.349,158.896
C04277=1025.672,170.703,387.311,168.702,47.353,158.897
C04278=1025.667,170.454,387.334,168.698,47.357,158.897
C04279=1025.660,170.205,387.356,168.695,47.361,158.898
C04280=1025.655,169.956,387.379,168.692,47.365,158.898
C04281=1025.649,169.707,387.401,168.689,47.369,158.898
C04282=1025.644,169.458,387.424,168.685,47.373,158.899
C04283=1025.638,169.210,387.446,168.681,47.377,158.899
C04284=1025.632,168.961,387.468,168.678,47.381,158.899
C04285=1025.627,168.712,387.491,168.674,47.385,158.900
C04286=1025.620,168.462,387.513,168.672,47.389,158.900
C04287=1025.615,168.214,387.535,168.668,47.393,158.900
C04288=1025.610,167.965,387.557,168.665,47.397,158.901
C04289=1025.604,167.716,387.580,168.661,47.401,158.901
C04290=1025.598,167.467,387.602,168.658,47.405,158.902
C04291=1025.593,167.218,387.624,168.654,47.409,158.902
C04292=1025.587,166.969,387.647,168.652,47.413,158.902
C04293=1025.581,166.720,387.669,168.648,47.417,158.903
C04294=1025.576,166.471,387.691,168.645,47.421,158.903
C04295=1025.570,166.223,387.714,168.641,47.425,158.903
C04296=1025.564,165.973,387.736,168.638,47.429,158.904
C04297=1025.559,165.724,387.758,168.635,47.433,158.904
C04298=1025.554,165.476,387.780,168.632,47.436,158.904
C04299=1025.548,165.227,387.802,168.628,47.441,158.905
C04300=1025.542,164.978,387.825,168.625,47.445,158.905
C04301=1025.537,164.729,387.847,168.621,47.449,158.906
C04302=1025.532,164.479,387.869,168.619,47.453,158.906
C04303=1025.525,164.231,387.891,168.616,47.456,158.906
C04304=1025.520,163.982,387.913,168.612,47.460,158.907
C04305=1025.515,163.733,387.936,168.609,47.465,158.907
C04306=1025.508,163.484,387.958,168.606,47.469,158.908
C04307=1025.504,163.235,387.980,168.603,47.473,158.908
C04308=1025.498,162.986,388.003,168.599,47.477,158.908
C04309=1025.492,162.737,388.024,168.596,47.480,158.909
C04310=1025.487,162.488,388.046,168.592,47.484,158.909
C04311=1025.481,162.239,388.069,168.589,47.488,158.909
C04312=1025.475,161.990,388.091,168.587,47.493,158.910
C04313=1025.470,161.741,388.113,168.583,47.497,158.910
C04314=1025.464,161.492,388.136,168.580,47.500,158.911
C04315=1025.459,161.244,388.157,168.576,47.504,158.911
C04316=1025.453,160.994,388.179,168.573,47.508,158.911
C04317=1025.448,160.745,388.201,168.570,47.512,158.912
C04318=1025.442,160.497,388.223,168.567,47.517,158.912
C04319=1025.437,160.247,388.245,168.564,47.520,158.912
C04320=1025.432,159.998,388.267,168.560,47.525,158.913
C04321=1025.426,159.749,388.289,168.557,47.528,158.913
C04322=1025.421,159.501,388.312,168.555,47.532,158.914
C04323=1025.415,159.252,388.334,168.551,47.536,158.914
C04324=1025.409,159.002,388.355,168.548,47.541,158.914
C04325=1025.403,158.754,388.377,168.544,47.545,158.915
C04326=1025.397,158.505,388.398,168.541,47.548,158.915
C04327=1025.392,158.255,388.421,168.538,47.553,158.916
C04328=1025.386,158.007,388.442,168.535,47.557,158.916
C04329=1025.380,157.757,388.463,168.532,47.562,158.916
C04330=1025.375,157.509,388.485,168.529,47.565,158.917
C04331=1025.369,157.259,388.507,168.525,47.569,158.917
C04332=1025.363,157.010,388.529,168.522,47.574,158.918
C04333=1025.357,156.762,388.550,168.519,47.578,158.918
C04334=1025.351,156.512,388.571,168.516,47.582,158.919
C04335=1025.346,156.229,388.596,168.512,47.587,158.919
C04336=1025.339,155.945,388.620,168.509,47.592,158.919
C04337=1025.332,155.662,388.645,168.505,47.596,158.920
C04338=1025.326,155.378,388.670,168.502,47.601,158.920
C04339=1025.320,155.129,388.691,168.498,47.605,158.921
C04340=1025.314,154.880,388.713,168.495,47.609,158.921
C04341=1025.309,154.631,388.734,168.493,47.613,158.922
C04342=1025.302,154.382,388.756,168.489,47.617,158.922
C04343=1025.298,154.133,388.777,168.486,47.621,158.922
C04344=1025.291,153.884,388.799,168.482,47.626,158.923
C04345=1025.286,153.636,388.820,168.479,47.630,158.923
C04346=1025.280,153.386,388.841,168.477,47.634,158.924
C04347=1025.274,153.137,388.863,168.473,47.638,158.924
C04348=1025.268,152.888,388.884,168.471,47.643,158.925
C04349=1025.263,152.639,388.906,168.467,47.647,158.925
C04350=1025.257,152.390,388.928,168.464,47.651,158.925
C04351=1025.252,152.141,388.948,168.460,47.655,158.926
C04352=1025.246,151.892,388.970,168.458,47.659,158.926
C04353=1025.240,151.643,388.991,168.455,47.664,158.927
C04354=1025.234,151.394,389.013,168.451,47.668,158.927
C04355=1025.229,151.145,389.033,168.449,47.672,158.928
C04356=1025.223,150.896,389.055,168.445,47.676,158.928
C04357=1025.217,150.647,389.076,168.442,47.681,158.928
C04358=1025.211,150.397,389.097,168.439,47.684,158.929
C04359=1025.206,150.149,389.118,168.436,47.688,158.929
C04360=1025.200,149.900,389.140,168.433,47.693,158.930
C04361=1025.194,149.651,389.161,168.429,47.697,158.930
C04362=1025.188,149.401,389.182,168.427,47.701,158.930
C04363=1025.183,149.153,389.203,168.424,47.705,158.931
C04364=1025.177,148.904,389.225,168.420,47.710,158.931
C04365=1025.171,148.655,389.246,168.418,47.714,158.932
C04366=1025.166,148.406,389.267,168.414,47.718,158.932
C04367=1025.160,148.156,389.288,168.411,47.722,158.933
C04368=1025.154,147.908,389.309,168.409,47.727,158.933
C04369=1025.148,147.659,389.331,168.405,47.731,158.933
C04370=1025.143,147.409,389.351,168.402,47.735,158.934
C04371=1025.137,147.161,389.373,168.399,47.739,158.934
C04372=1025.131,146.911,389.393,168.396,47.743,158.935
C04373=1025.126,146.663,389.415,168.393,47.748,158.935
C04374=1025.120,146.413,389.436,168.389,47.752,158.935
C04375=1025.114,146.164,389.457,168.387,47.756,158.936
C04376=1025.109,145.915,389.478,168.384,47.760,158.936
C04377=1025.103,145.666,389.499,168.380,47.765,158.937
C04378=1025.098,145.417,389.520,168.378,47.769,158.937
C04379=1025.091,145.168,389.541,168.375,47.773,158.938
C04380=1025.086,144.919,389.561,168.372,47.778,158.938
C04381=1025.080,144.670,389.583,168.369,47.781,158.939
C04382=1025.074,144.420,389.603,168.365,47.786,158.939
C04383=1025.069,144.172,389.625,168.362,47.790,158.939
C04384=1025.063,143.923,389.645,168.360,47.794,158.940
C04385=1025.057,143.673,389.666,168.356,47.799,158.940
C04386=1025.051,143.425,389.687,168.354,47.803,158.941
C04387=1025.045,143.175,389.708,168.351,47.807,158.941
C04388=1025.040,142.926,389.729,168.347,47.812,158.942
C04389=1025.034,142.678,389.749,168.345,47.816,158.942
C04390=1025.028,142.428,389.770,168.341,47.820,158.943
C04391=1025.022,142.179,389.791,168.338,47.825,158.943
C04392=1025.017,141.930,389.812,168.336,47.828,158.943
C04393=1025.011,141.680,389.833,168.332,47.833,158.944
C04394=1025.005,141.432,389.853,168.329,47.837,158.944
C04395=1025.000,141.183,389.874,168.327,47.841,158.945
C04396=1024.994,140.934,389.894,168.323,47.846,158.945
C04397=1024.988,140.685,389.916,168.320,47.850,158.946
C04398=1024.982,140.436,389.936,168.318,47.855,158.946
C04399=1024.975,140.152,389.960,168.314,47.859,158.947
C04400=1024.970,139.868,389.983,168.311,47.864,158.947
C04401=1024.963,139.584,390.007,168.307,47.869,158.948
C04402=1024.957,139.300,390.031,168.304,47.874,158.948
C04403=1024.951,139.051,390.052,168.301,47.878,158.949
C04404=1024.945,138.802,390.072,168.297,47.882,158.949
C04405=1024.939,138.553,390.093,168.295,47.887,158.950
C04406=1024.934,138.304,390.113,168.292,47.890,158.950
C04407=1024.928,138.054,390.134,168.289,47.895,158.950
C04408=1024.922,137.806,390.154,168.286,47.900,158.951
C04409=1024.917,137.556,390.175,168.283,47.903,158.951
C04410=1024.910,137.308,390.196,168.280,47.908,158.952
C04411=1024.905,137.058,390.216,168.277,47.912,158.952
C04412=1024.900,136.809,390.237,168.274,47.917,158.953
C04413=1024.894,136.560,390.257,168.272,47.921,158.953
C04414=1024.888,136.311,390.278,168.268,47.925,158.954
C04415=1024.882,136.062,390.298,168.266,47.930,158.954
C04416=1024.877,135.813,390.318,168.263,47.934,158.955
C04417=1024.871,135.564,390.338,168.259,47.938,158.955
C04418=1024.865,135.315,390.359,168.257,47.943,158.955
C04419=1024.859,135.065,390.379,168.254,47.947,158.956
C04420=1024.853,134.817,390.400,168.250,47.951,158.956
C04421=1024.847,134.568,390.420,168.248,47.956,158.957
C04422=1024.842,134.319,390.441,168.245,47.960,158.957
C04423=1024.835,134.069,390.461,168.242,47.964,158.958
C04424=1024.830,133.820,390.482,168.239,47.969,158.958
C04425=1024.824,133.571,390.502,168.236,47.973,158.959
C04426=1024.819,133.322,390.522,168.233,47.977,158.959
C04427=1024.814,133.073,390.543,168.230,47.982,158.960
C04428=1024.807,132.824,390.563,168.228,47.986,158.960
C04429=1024.802,132.574,390.584,168.225,47.990,158.961
C04430=1024.796,132.326,390.604,168.221,47.994,158.961
C04431=1024.790,132.077,390.624,168.219,47.999,158.961
C04432=1024.785,131.827,390.644,168.216,48.003,158.962
C04433=1024.779,131.578,390.664,168.212,48.008,158.962
C04434=1024.773,131.328,390.684,168.210,48.012,158.963
C04435=1024.768,131.079,390.705,168.207,48.017,158.963
C04436=1024.762,130.831,390.725,168.205,48.020,158.964
C04437=1024.756,130.581,390.745,168.201,48.025,158.964
C04438=1024.750,130.333,390.765,168.198,48.029,158.964
C04439=1024.744,130.084,390.785,168.196,48.033,158.965
C04440=1024.739,129.835,390.806,168.192,48.038,158.965
C04441=1024.733,129.585,390.826,168.190,48.043,158.966
C04442=1024.727,129.336,390.846,168.187,48.047,158.966
C04443=1024.721,129.087,390.865,168.184,48.051,158.967
C04444=1024.715,128.838,390.885,168.181,48.056,158.967
C04445=1024.709,128.589,390.905,168.179,48.060,158.968
C04446=1024.704,128.340,390.925,168.175,48.065,158.968
C04447=1024.697,128.090,390.946,168.172,48.069,158.969
C04448=1024.691,127.841,390.966,168.170,48.074,158.969
C04449=1024.686,127.592,390.985,168.166,48.078,158.970
C04450=1024.680,127.343,391.005,168.164,48.083,158.970
C04451=1024.674,127.094,391.025,168.161,48.087,158.971
C04452=1024.669,126.844,391.045,168.159,48.091,158.971
C04453=1024.663,126.596,391.064,168.155,48.096,158.972
C04454=1024.657,126.347,391.084,168.153,48.100,158.972
C04455=1024.651,126.097,391.104,168.150,48.104,158.973
C04456=1024.644,125.848,391.124,168.146,48.109,158.973
C04457=1024.638,125.599,391.144,168.144,48.114,158.974
C04458=1024.634,125.349,391.164,168.141,48.118,158.974
C04459=1024.628,125.100,391.184,168.138,48.122,158.974
C04460=1024.622,124.852,391.204,168.135,48.127,158.975
C04461=1024.616,124.602,391.223,168.133,48.131,158.976
C04462=1024.610,124.353,391.243,168.130,48.136,158.976
C04463=1024.603,124.070,391.265,168.127,48.141,158.977
C04464=1024.597,123.785,391.289,168.123,48.146,158.977
C04465=1024.590,123.501,391.311,168.120,48.151,158.978
C04466=1024.584,123.218,391.333,168.116,48.156,158.978
C04467=1024.578,122.968,391.352,168.114,48.160,158.979
C04468=1024.572,122.720,391.372,168.111,48.165,158.979
C04469=1024.566,122.471,391.392,168.108,48.170,158.980
C04470=1024.561,122.221,391.412,168.105,48.173,158.980
C04471=1024.555,121.972,391.432,168.103,48.178,158.981
C04472=1024.549,121.722,391.452,168.100,48.182,158.981
C04473=1024.543,121.473,391.472,168.096,48.187,158.981
C04474=1024.537,121.224,391.491,168.094,48.191,158.982
C04475=1024.531,120.975,391.511,168.091,48.196,158.982
C04476=1024.526,120.726,391.530,168.089,48.200,158.983
C04477=1024.520,120.476,391.551,168.085,48.204,158.983
C04478=1024.515,120.227,391.570,168.083,48.209,158.984
C04479=1024.509,119.978,391.590,168.080,48.213,158.984
C04480=1024.503,119.729,391.609,168.077,48.217,158.985
C04481=1024.497,119.481,391.629,168.074,48.222,158.985
C04482=1024.492,119.231,391.648,168.072,48.227,158.986
C04483=1024.486,118.982,391.668,168.069,48.230,158.986
C04484=1024.481,118.733,391.688,168.066,48.235,158.987
C04485=1024.475,118.484,391.708,168.064,48.239,158.987
C04486=1024.469,118.234,391.727,168.060,48.244,158.987
C04487=1024.463,117.986,391.747,168.058,48.248,158.988
C04488=1024.457,117.736,391.766,168.055,48.253,158.989
C04489=1024.452,117.487,391.785,168.053,48.257,158.989
C04490=1024.446,117.238,391.805,168.050,48.261,158.989
C04491=1024.440,116.988,391.825,168.046,48.266,158.990
C04492=1024.435,116.739,391.845,168.044,48.270,158.990
C04493=1024.429,116.490,391.864,168.041,48.274,158.991
C04494=1024.423,116.240,391.884,168.039,48.279,158.991
C04495=1024.418,115.992,391.904,168.036,48.283,158.992
C04496=1024.412,115.742,391.923,168.032,48.287,158.992
C04497=1024.406,115.494,391.942,168.030,48.292,158.993
C04498=1024.401,115.245,391.962,168.027,48.296,158.993
C04499=1024.395,114.995,391.981,168.025,48.300,158.994
C04500=1024.390,114.746,392.002,168.022,48.305,158.994
C04501=1024.384,114.497,392.021,168.019,48.309,158.995
C04502=1024.378,114.247,392.040,168.016,48.314,158.995
C04503=1024.372,113.998,392.060,168.013,48.318,158.996
C04504=1024.367,113.749,392.079,168.011,48.322,158.996
C04505=1024.362,113.500,392.098,168.008,48.327,158.996
C04506=1024.356,113.251,392.118,168.006,48.331,158.997
C04507=1024.350,113.002,392.137,168.003,48.335,158.997
C04508=1024.345,112.752,392.157,168.001,48.340,158.998
C04509=1024.339,112.503,392.176,167.997,48.344,158.998
C04510=1024.333,112.254,392.196,167.994,48.348,158.999
C04511=1024.327,112.005,392.215,167.992,48.353,158.999
C04512=1024.321,111.755,392.234,167.989,48.357,159.000
C04513=1024.316,111.506,392.253,167.986,48.362,159.000
C04514=1024.310,111.257,392.272,167.983,48.366,159.001
C04515=1024.305,111.008,392.292,167.981,48.371,159.001
C04516=1024.298,110.759,392.311,167.978,48.375,159.002
C04517=1024.292,110.510,392.330,167.976,48.380,159.002
C04518=1024.287,110.261,392.349,167.972,48.384,159.002
C04519=1024.281,110.011,392.369,167.969,48.388,159.003
C04520=1024.275,109.762,392.388,167.967,48.393,159.004
C04521=1024.269,109.513,392.406,167.965,48.398,159.004
C04522=1024.264,109.264,392.425,167.962,48.402,159.005
C04523=1024.258,109.014,392.445,167.958,48.406,159.005
C04524=1024.252,108.765,392.463,167.956,48.411,159.005
C04525=1024.246,108.516,392.483,167.953,48.415,159.006
C04526=1024.240,108.266,392.502,167.951,48.420,159.007
C04527=1024.233,107.982,392.523,167.948,48.425,159.007
C04528=1024.227,107.699,392.545,167.944,48.430,159.008
C04529=1024.221,107.414,392.567,167.941,48.435,159.008
C04530=1024.214,107.131,392.588,167.938,48.441,159.009
C04531=1024.208,106.881,392.607,167.935,48.445,159.009
C04532=1024.202,106.632,392.626,167.933,48.450,159.010
C04533=1024.196,106.383,392.645,167.930,48.454,159.010
C04534=1024.191,106.134,392.664,167.928,48.458,159.011
C04535=1024.184,105.885,392.682,167.924,48.463,159.011
C04536=1024.179,105.635,392.702,167.922,48.468,159.012
C04537=1024.173,105.386,392.721,167.919,48.472,159.012
C04538=1024.167,105.137,392.739,167.917,48.476,159.013
C04539=1024.161,104.888,392.758,167.914,48.481,159.013
C04540=1024.156,104.639,392.778,167.911,48.485,159.014
C04541=1024.150,104.389,392.796,167.908,48.490,159.014
C04542=1024.144,104.140,392.815,167.906,48.495,159.015
C04543=1024.139,103.891,392.834,167.903,48.498,159.015
C04544=1024.132,103.642,392.852,167.901,48.503,159.016
C04545=1024.127,103.392,392.872,167.898,48.508,159.016
C04546=1024.122,103.143,392.891,167.895,48.512,159.017
C04547=1024.115,102.894,392.909,167.892,48.516,159.017
C04548=1024.109,102.645,392.928,167.889,48.521,159.017
C04549=1024.104,102.395,392.947,167.887,48.525,159.018
C04550=1024.098,102.146,392.965,167.885,48.530,159.019
C04551=1024.093,101.897,392.984,167.882,48.535,159.019
C04552=1024.086,101.648,393.003,167.878,48.539,159.019
C04553=1024.081,101.399,393.022,167.876,48.543,159.020
C04554=1024.075,101.150,393.041,167.873,48.548,159.020
C04555=1024.069,100.900,393.059,167.871,48.552,159.021
C04556=1024.064,100.650,393.078,167.868,48.556,159.021
C04557=1024.058,100.402,393.097,167.866,48.561,159.022
C04558=1024.052,100.153,393.116,167.863,48.566,159.022
C04559=1024.046,99.903,393.135,167.860,48.570,159.023
C04560=1024.042,99.654,393.153,167.857,48.574,159.023
C04561=1024.035,99.405,393.172,167.855,48.579,159.024
C04562=1024.029,99.156,393.191,167.852,48.583,159.024
C04563=1024.024,98.906,393.209,167.850,48.588,159.025
C04564=1024.017,98.657,393.227,167.846,48.593,159.025
C04565=1024.011,98.408,393.246,167.844,48.597,159.026
C04566=1024.006,98.158,393.265,167.841,48.601,159.026
C04567=1024.000,97.909,393.283,167.839,48.606,159.027
C04568=1023.994,97.659,393.301,167.836,48.610,159.027
C04569=1023.988,97.410,393.320,167.833,48.615,159.028
C04570=1023.982,97.162,393.338,167.830,48.620,159.028
C04571=1023.977,96.912,393.357,167.828,48.625,159.029
C04572=1023.970,96.663,393.376,167.826,48.629,159.029
C04573=1023.965,96.414,393.393,167.823,48.633,159.030
C04574=1023.959,96.164,393.412,167.819,48.638,159.030
C04575=1023.953,95.915,393.431,167.817,48.642,159.031
C04576=1023.947,95.666,393.449,167.815,48.647,159.031
C04577=1023.942,95.417,393.468,167.812,48.652,159.032
C04578=1023.935,95.167,393.486,167.810,48.656,159.032
C04579=1023.930,94.918,393.504,167.807,48.660,159.033
C04580=1023.924,94.668,393.523,167.803,48.665,159.033
C04581=1023.918,94.420,393.541,167.801,48.670,159.034
C04582=1023.912,94.170,393.559,167.799,48.674,159.034
C04583=1023.907,93.921,393.578,167.796,48.679,159.035
C04584=1023.901,93.672,393.596,167.793,48.683,159.035
C04585=1023.895,93.423,393.614,167.791,48.687,159.036
C04586=1023.889,93.173,393.633,167.788,48.692,159.036
C04587=1023.883,92.924,393.651,167.785,48.697,159.036
C04588=1023.877,92.674,393.669,167.783,48.701,159.037
C04589=1023.872,92.426,393.688,167.780,48.705,159.037
C04590=1023.866,92.176,393.706,167.778,48.710,159.038
C04591=1023.859,91.892,393.727,167.774,48.715,159.039
C04592=1023.853,91.609,393.747,167.771,48.720,159.039
C04593=1023.847,91.324,393.769,167.769,48.726,159.040
C04594=1023.840,91.040,393.789,167.765,48.730,159.040
C04595=1023.834,90.791,393.808,167.763,48.735,159.041
C04596=1023.829,90.541,393.826,167.761,48.740,159.041
C04597=1023.823,90.293,393.844,167.758,48.744,159.042
C04598=1023.817,90.043,393.862,167.754,48.748,159.042
C04599=1023.812,89.794,393.881,167.752,48.753,159.043
C04600=1023.805,89.545,393.899,167.750,48.758,159.043
C04601=1023.799,89.295,393.917,167.747,48.761,159.043
C04602=1023.794,89.046,393.935,167.744,48.766,159.044
C04603=1023.787,88.797,393.953,167.742,48.771,159.044
C04604=1023.782,88.548,393.971,167.739,48.776,159.045
C04605=1023.776,88.298,393.989,167.736,48.780,159.045
C04606=1023.770,88.050,394.007,167.734,48.785,159.046
C04607=1023.764,87.800,394.025,167.731,48.789,159.047
C04608=1023.758,87.550,394.043,167.729,48.794,159.047
C04609=1023.752,87.301,394.061,167.725,48.799,159.048
C04610=1023.746,87.051,394.078,167.723,48.803,159.048
C04611=1023.741,86.803,394.097,167.720,48.807,159.048
C04612=1023.735,86.553,394.115,167.718,48.812,159.049
C04613=1023.729,86.304,394.133,167.716,48.817,159.049
C04614=1023.723,86.054,394.151,167.713,48.821,159.050
C04615=1023.717,85.806,394.169,167.710,48.826,159.050
C04616=1023.711,85.556,394.187,167.707,48.831,159.051
C04617=1023.706,85.307,394.205,167.705,48.835,159.052
C04618=1023.700,85.057,394.223,167.702,48.840,159.052
C04619=1023.694,84.808,394.240,167.700,48.844,159.052
C04620=1023.688,84.558,394.258,167.696,48.849,159.053
C04621=1023.682,84.310,394.276,167.694,48.853,159.053
C04622=1023.676,84.060,394.294,167.691,48.858,159.054
C04623=1023.671,83.811,394.312,167.689,48.863,159.054
C04624=1023.664,83.561,394.330,167.687,48.867,159.055
C04625=1023.659,83.312,394.347,167.684,48.871,159.055
C04626=1023.653,83.063,394.365,167.681,48.876,159.056
C04627=1023.647,82.814,394.383,167.678,48.881,159.056
C04628=1023.641,82.564,394.401,167.676,48.885,159.057
C04629=1023.635,82.316,394.419,167.673,48.890,159.057
C04630=1023.630,82.066,394.437,167.671,48.894,159.058
C04631=1023.624,81.817,394.455,167.668,48.898,159.058
C04632=1023.618,81.568,394.472,167.666,48.903,159.059
C04633=1023.612,81.318,394.490,167.663,48.908,159.059
C04634=1023.607,81.069,394.508,167.660,48.913,159.060
C04635=1023.600,80.819,394.526,167.657,48.917,159.060
C04636=1023.595,80.570,394.543,167.655,48.921,159.061
C04637=1023.589,80.320,394.561,167.652,48.926,159.061
C04638=1023.583,80.071,394.579,167.650,48.930,159.062
C04639=1023.578,79.822,394.596,167.648,48.935,159.062
C04640=1023.572,79.573,394.614,167.645,48.940,159.063
C04641=1023.566,79.324,394.632,167.641,48.944,159.063
C04642=1023.560,79.074,394.650,167.639,48.948,159.064
C04643=1023.554,78.825,394.667,167.637,48.953,159.064
C04644=1023.549,78.576,394.685,167.634,48.958,159.065
C04645=1023.543,78.326,394.703,167.631,48.962,159.065
C04646=1023.537,78.077,394.720,167.629,48.966,159.066
C04647=1023.532,77.828,394.738,167.627,48.971,159.066
C04648=1023.526,77.578,394.756,167.624,48.975,159.067
C04649=1023.520,77.329,394.773,167.622,48.979,159.067
C04650=1023.514,77.079,394.791,167.618,48.984,159.067
C04651=1023.508,76.831,394.808,167.616,48.989,159.068
C04652=1023.502,76.582,394.826,167.613,48.994,159.068
C04653=1023.496,76.332,394.844,167.611,48.998,159.069
C04654=1023.491,76.083,394.861,167.609,49.003,159.069
C04655=1023.483,75.799,394.881,167.605,49.008,159.070
C04656=1023.477,75.515,394.901,167.602,49.013,159.071
C04657=1023.470,75.230,394.921,167.600,49.018,159.071
C04658=1023.464,74.947,394.941,167.597,49.024,159.072
C04659=1023.458,74.697,394.958,167.594,49.028,159.072
C04660=1023.451,74.448,394.975,167.591,49.033,159.073
C04661=1023.446,74.198,394.992,167.588,49.037,159.073
C04662=1023.441,73.949,395.010,167.586,49.042,159.074
C04663=1023.434,73.700,395.028,167.583,49.046,159.074
C04664=1023.428,73.451,395.045,167.581,49.051,159.075
C04665=1023.423,73.202,395.062,167.578,49.056,159.075
C04666=1023.417,72.951,395.080,167.576,49.060,159.076
C04667=1023.411,72.703,395.097,167.572,49.064,159.076
C04668=1023.405,72.454,395.114,167.570,49.069,159.076
C04669=1023.399,72.204,395.132,167.568,49.074,159.077
C04670=1023.394,71.954,395.149,167.565,49.078,159.077
C04671=1023.387,71.706,395.166,167.563,49.083,159.078
C04672=1023.381,71.456,395.184,167.560,49.088,159.079
C04673=1023.376,71.206,395.201,167.558,49.092,159.079
C04674=1023.370,70.957,395.218,167.554,49.097,159.079
C04675=1023.364,70.708,395.235,167.552,49.101,159.080
C04676=1023.358,70.459,395.253,167.549,49.106,159.080
C04677=1023.352,70.209,395.269,167.547,49.110,159.081
C04678=1023.347,69.960,395.287,167.544,49.114,159.081
C04679=1023.341,69.711,395.305,167.542,49.119,159.082
C04680=1023.335,69.461,395.321,167.540,49.124,159.082
C04681=1023.329,69.212,395.339,167.536,49.129,159.083
C04682=1023.324,68.963,395.356,167.534,49.133,159.083
C04683=1023.317,68.713,395.373,167.531,49.137,159.084
C04684=1023.312,68.464,395.390,167.529,49.142,159.084
C04685=1023.306,68.214,395.407,167.526,49.147,159.085
C04686=1023.300,67.966,395.424,167.524,49.151,159.085
C04687=1023.294,67.716,395.442,167.521,49.156,159.086
C04688=1023.288,67.467,395.458,167.518,49.161,159.086
C04689=1023.283,67.217,395.476,167.515,49.165,159.087
C04690=1023.276,66.967,395.493,167.513,49.169,159.087
C04691=1023.270,66.718,395.510,167.511,49.174,159.088
C04692=1023.265,66.469,395.526,167.508,49.179,159.088
C04693=1023.259,66.220,395.544,167.506,49.183,159.089
C04694=1023.253,65.971,395.560,167.503,49.188,159.089
C04695=1023.247,65.721,395.578,167.500,49.192,159.089
C04696=1023.241,65.472,395.594,167.497,49.197,159.090
C04697=1023.235,65.223,395.612,167.495,49.201,159.090
C04698=1023.229,64.973,395.628,167.493,49.206,159.091
C04699=1023.223,64.723,395.646,167.490,49.211,159.092
C04700=1023.217,64.474,395.662,167.487,49.216,159.092
C04701=1023.212,64.225,395.680,167.484,49.220,159.092
C04702=1023.206,63.976,395.696,167.482,49.224,159.093
C04703=1023.201,63.726,395.713,167.479,49.229,159.093
C04704=1023.194,63.477,395.730,167.477,49.234,159.094
C04705=1023.189,63.227,395.747,167.475,49.238,159.094
C04706=1023.182,62.978,395.764,167.471,49.243,159.095
C04707=1023.176,62.729,395.781,167.469,49.248,159.095
C04708=1023.170,62.479,395.797,167.467,49.253,159.096
C04709=1023.165,62.229,395.814,167.464,49.257,159.096
C04710=1023.158,61.980,395.831,167.462,49.262,159.097
C04711=1023.152,61.731,395.847,167.458,49.267,159.097
C04712=1023.147,61.482,395.864,167.456,49.272,159.098
C04713=1023.140,61.232,395.881,167.453,49.275,159.098
C04714=1023.134,60.983,395.897,167.451,49.280,159.099
C04715=1023.129,60.733,395.914,167.448,49.285,159.099
C04716=1023.123,60.484,395.930,167.445,49.290,159.100
C04717=1023.116,60.235,395.947,167.443,49.294,159.100
C04718=1023.110,59.985,395.964,167.441,49.299,159.101
C04719=1023.103,59.701,395.982,167.437,49.305,159.101
C04720=1023.097,59.417,396.001,167.434,49.310,159.102
C04721=1023.090,59.133,396.020,167.431,49.315,159.102
C04722=1023.083,58.848,396.039,167.429,49.321,159.103
C04723=1023.077,58.599,396.056,167.426,49.326,159.104
C04724=1023.071,58.350,396.072,167.423,49.330,159.104
C04725=1023.065,58.101,396.089,167.421,49.334,159.104
C04726=1023.059,57.852,396.105,167.418,49.339,159.105
C04727=1023.054,57.602,396.122,167.415,49.344,159.105
C04728=1023.048,57.353,396.138,167.412,49.349,159.106
C04729=1023.042,57.103,396.155,167.410,49.353,159.106
C04730=1023.035,56.853,396.171,167.408,49.358,159.107
C04731=1023.029,56.604,396.188,167.405,49.363,159.108
C04732=1023.023,56.355,396.204,167.403,49.367,159.108
C04733=1023.018,56.105,396.221,167.400,49.372,159.108
C04734=1023.012,55.856,396.237,167.397,49.376,159.109
C04735=1023.006,55.607,396.254,167.395,49.381,159.109
C04736=1023.000,55.357,396.270,167.392,49.386,159.110
C04737=1022.994,55.108,396.286,167.390,49.390,159.110
C04738=1022.988,54.859,396.303,167.386,49.395,159.111
C04739=1022.982,54.610,396.320,167.384,49.400,159.111
C04740=1022.976,54.360,396.336,167.381,49.404,159.112
C04741=1022.970,54.110,396.353,167.379,49.409,159.112
C04742=1022.964,53.861,396.369,167.377,49.413,159.113
C04743=1022.958,53.612,396.385,167.374,49.418,159.113
C04744=1022.952,53.362,396.402,167.371,49.423,159.114
C04745=1022.946,53.113,396.418,167.369,49.428,159.114
C04746=1022.941,52.863,396.435,167.366,49.432,159.115
C04747=1022.935,52.614,396.451,167.364,49.436,159.115
C04748=1022.929,52.364,396.467,167.361,49.441,159.116
C04749=1022.923,52.115,396.484,167.359,49.446,159.116
C04750=1022.917,51.866,396.500,167.356,49.451,159.117
C04751=1022.911,51.616,396.516,167.353,49.455,159.117
C04752=1022.905,51.367,396.532,167.350,49.459,159.117
C04753=1022.900,51.117,396.549,167.348,49.464,159.118
C04754=1022.894,50.868,396.565,167.346,49.469,159.118
C04755=1022.888,50.619,396.582,167.343,49.473,159.119
C04756=1022.882,50.369,396.598,167.340,49.478,159.119
C04757=1022.876,50.120,396.614,167.337,49.482,159.120
C04758=1022.870,49.871,396.630,167.335,49.487,159.120
C04759=1022.864,49.621,396.647,167.332,49.491,159.121
C04760=1022.859,49.372,396.664,167.330,49.496,159.121
C04761=1022.853,49.122,396.680,167.328,49.500,159.122
C04762=1022.847,48.873,396.696,167.325,49.505,159.122
C04763=1022.841,48.624,396.712,167.322,49.509,159.122
C04764=1022.835,48.374,396.729,167.319,49.514,159.123
C04765=1022.829,48.125,396.745,167.317,49.519,159.123
C04766=1022.823,47.876,396.761,167.314,49.523,159.124
C04767=1022.817,47.626,396.777,167.312,49.527,159.124
C04768=1022.812,47.377,396.794,167.309,49.532,159.125
C04769=1022.806,47.127,396.810,167.307,49.537,159.125
C04770=1022.800,46.878,396.827,167.303,49.541,159.126
C04771=1022.795,46.629,396.843,167.301,49.546,159.126
C04772=1022.789,46.379,396.858,167.299,49.550,159.127
C04773=1022.783,46.130,396.874,167.296,49.554,159.127
C04774=1022.777,45.881,396.891,167.294,49.559,159.128
C04775=1022.772,45.631,396.908,167.291,49.564,159.128
C04776=1022.766,45.382,396.924,167.289,49.568,159.128
C04777=1022.760,45.132,396.940,167.286,49.573,159.129
C04778=1022.754,44.883,396.956,167.284,49.577,159.129
C04779=1022.749,44.633,396.972,167.280,49.582,159.130
C04780=1022.743,44.384,396.988,167.278,49.586,159.130
C04781=1022.737,44.134,397.004,167.276,49.591,159.131
C04782=1022.731,43.886,397.020,167.273,49.595,159.131
C04783=1022.724,43.601,397.039,167.269,49.600,159.131
C04784=1022.718,43.316,397.057,167.268,49.605,159.132
C04785=1022.712,43.032,397.076,167.264,49.610,159.133
C04786=1022.705,42.747,397.094,167.261,49.615,159.133
C04787=1022.699,42.498,397.111,167.258,49.620,159.134
C04788=1022.694,42.249,397.126,167.256,49.625,159.134
C04789=1022.688,41.999,397.142,167.253,49.629,159.134
C04790=1022.682,41.750,397.158,167.251,49.633,159.135
C04791=1022.676,41.500,397.173,167.249,49.638,159.135
C04792=1022.670,41.251,397.190,167.245,49.643,159.136
C04793=1022.664,41.002,397.206,167.243,49.648,159.136
C04794=1022.658,40.752,397.221,167.240,49.652,159.137
C04795=1022.652,40.502,397.238,167.238,49.657,159.137
C04796=1022.647,40.254,397.253,167.236,49.661,159.138
C04797=1022.641,40.004,397.268,167.232,49.666,159.138
C04798=1022.635,39.755,397.285,167.230,49.670,159.139
C04799=1022.629,39.505,397.300,167.227,49.675,159.139
C04800=1022.623,39.255,397.316,167.225,49.680,159.140
C04801=1022.617,39.006,397.333,167.222,49.684,159.140
C04802=1022.612,38.757,397.348,167.220,49.688,159.140
C04803=1022.605,38.508,397.364,167.217,49.693,159.141
C04804=1022.600,38.258,397.379,167.214,49.698,159.141
C04805=1022.594,38.009,397.395,167.212,49.702,159.142
C04806=1022.588,37.759,397.412,167.209,49.707,159.142
C04807=1022.582,37.509,397.427,167.207,49.712,159.143
C04808=1022.577,37.261,397.443,167.204,49.716,159.143
C04809=1022.570,37.011,397.458,167.202,49.720,159.144
C04810=1022.564,36.762,397.474,167.199,49.725,159.144
C04811=1022.559,36.512,397.490,167.196,49.729,159.144
C04812=1022.552,36.262,397.505,167.194,49.734,159.145
C04813=1022.546,36.013,397.521,167.191,49.739,159.145
C04814=1022.541,35.763,397.536,167.188,49.744,159.146
C04815=1022.535,35.514,397.552,167.186,49.748,159.146
C04816=1022.529,35.264,397.567,167.183,49.753,159.147
C04817=1022.523,35.015,397.582,167.181,49.757,159.147
C04818=1022.517,34.765,397.599,167.178,49.762,159.148
C04819=1022.512,34.516,397.614,167.175,49.767,159.148
C04820=1022.505,34.267,397.629,167.173,49.772,159.149
C04821=1022.499,34.017,397.645,167.170,49.776,159.149
C04822=1022.493,33.767,397.660,167.168,49.780,159.149
C04823=1022.488,33.519,397.676,167.164,49.785,159.150
C04824=1022.482,33.269,397.691,167.162,49.790,159.150
C04825=1022.476,33.019,397.706,167.160,49.795,159.151
C04826=1022.470,32.770,397.723,167.157,49.799,159.151
C04827=1022.464,32.521,397.737,167.155,49.804,159.152
C04828=1022.458,32.271,397.753,167.151,49.809,159.152
C04829=1022.452,32.022,397.768,167.149,49.813,159.153
C04830=1022.446,31.772,397.784,167.146,49.817,159.153
C04831=1022.441,31.523,397.799,167.144,49.822,159.154
C04832=1022.434,31.274,397.815,167.142,49.827,159.154
C04833=1022.429,31.024,397.830,167.138,49.831,159.154
C04834=1022.423,30.775,397.845,167.136,49.836,159.155
C04835=1022.417,30.525,397.861,167.133,49.841,159.155
C04836=1022.410,30.276,397.876,167.131,49.845,159.156
C04837=1022.405,30.026,397.892,167.128,49.849,159.156
C04838=1022.400,29.776,397.907,167.125,49.854,159.157
C04839=1022.393,29.527,397.922,167.123,49.859,159.157
C04840=1022.387,29.277,397.938,167.120,49.863,159.157
C04841=1022.382,29.028,397.953,167.118,49.868,159.158
C04842=1022.376,28.778,397.968,167.115,49.873,159.158
C04843=1022.369,28.529,397.984,167.113,49.877,159.159
C04844=1022.364,28.280,397.999,167.109,49.882,159.159
C04845=1022.359,28.030,398.014,167.107,49.886,159.160
C04846=1022.352,27.781,398.029,167.104,49.890,159.160
C04847=1022.345,27.496,398.047,167.101,49.896,159.161
C04848=1022.339,27.212,398.064,167.098,49.901,159.161
C04849=1022.332,26.928,398.081,167.095,49.906,159.161
C04850=1022.326,26.643,398.099,167.093,49.912,159.162
C04851=1022.319,26.393,398.114,167.089,49.917,159.163
C04852=1022.314,26.144,398.128,167.087,49.921,159.163
C04853=1022.308,25.894,398.144,167.085,49.926,159.163
C04854=1022.301,25.645,398.160,167.082,49.930,159.164
C04855=1022.295,25.396,398.174,167.080,49.935,159.165
C04856=1022.290,25.146,398.190,167.076,49.939,159.165
C04857=1022.284,24.897,398.204,167.074,49.944,159.165
C04858=1022.278,24.648,398.219,167.072,49.949,159.166
C04859=1022.272,24.398,398.235,167.069,49.954,159.166
C04860=1022.266,24.149,398.249,167.066,49.958,159.166
C04861=1022.260,23.899,398.264,167.063,49.963,159.167
C04862=1022.254,23.649,398.280,167.061,49.967,159.168
C04863=1022.248,23.400,398.294,167.058,49.971,159.168
C04864=1022.242,23.151,398.309,167.055,49.976,159.168
C04865=1022.237,22.901,398.325,167.053,49.981,159.169
C04866=1022.231,22.652,398.340,167.050,49.986,159.169
C04867=1022.224,22.402,398.354,167.048,49.990,159.170
C04868=1022.219,22.153,398.370,167.044,49.995,159.170
C04869=1022.213,21.903,398.385,167.042,50.000,159.171
C04870=1022.207,21.654,398.399,167.039,50.004,159.171
C04871=1022.201,21.404,398.415,167.037,50.009,159.171
C04872=1022.196,21.155,398.429,167.035,50.013,159.172
C04873=1022.189,20.906,398.444,167.031,50.018,159.172
C04874=1022.184,20.655,398.459,167.029,50.022,159.173
C04875=1022.178,20.406,398.474,167.027,50.027,159.173
C04876=1022.172,20.156,398.489,167.024,50.031,159.173
C04877=1022.166,19.907,398.503,167.021,50.036,159.174
C04878=1022.160,19.657,398.519,167.018,50.041,159.174
C04879=1022.155,19.408,398.533,167.016,50.045,159.175
C04880=1022.148,19.159,398.548,167.013,50.050,159.175
C04881=1022.143,18.910,398.563,167.011,50.055,159.176
C04882=1022.137,18.660,398.578,167.007,50.059,159.176
C04883=1022.131,18.410,398.592,167.005,50.064,159.177
C04884=1022.125,18.161,398.607,167.003,50.068,159.177
C04885=1022.118,17.911,398.622,166.999,50.073,159.177
C04886=1022.113,17.662,398.637,166.997,50.078,159.178
C04887=1022.107,17.412,398.652,166.994,50.082,159.178
C04888=1022.102,17.162,398.666,166.992,50.086,159.179
C04889=1022.095,16.913,398.681,166.988,50.091,159.179
C04890=1022.089,16.664,398.696,166.986,50.096,159.180
C04891=1022.083,16.414,398.711,166.984,50.101,159.180
C04892=1022.078,16.165,398.724,166.981,50.105,159.180
C04893=1022.072,15.915,398.740,166.978,50.110,159.181
C04894=1022.066,15.666,398.755,166.975,50.114,159.181
C04895=1022.060,15.417,398.769,166.973,50.119,159.182
C04896=1022.054,15.166,398.783,166.971,50.124,159.182
C04897=1022.048,14.918,398.798,166.968,50.128,159.182
C04898=1022.042,14.668,398.813,166.965,50.133,159.183
C04899=1022.036,14.419,398.827,166.962,50.138,159.183
C04900=1022.031,14.168,398.842,166.960,50.142,159.184
C04901=1022.025,13.919,398.857,166.957,50.146,159.184
C04902=1022.019,13.670,398.872,166.954,50.151,159.185
C04903=1022.013,13.420,398.886,166.952,50.156,159.185
C04904=1022.007,13.170,398.901,166.949,50.160,159.185
C04905=1022.001,12.921,398.914,166.946,50.165,159.186
C04906=1021.995,12.671,398.929,166.943,50.169,159.186
C04907=1021.990,12.422,398.943,166.941,50.174,159.187
C04908=1021.983,12.173,398.957,166.938,50.179,159.187
C04909=1021.977,11.923,398.972,166.935,50.184,159.188
C04910=1021.971,11.674,398.986,166.933,50.189,159.188
C04911=1021.966,11.456,398.999,166.930,50.193,159.188
C04912=1021.960,11.240,399.011,166.928,50.197,159.189
C04913=1021.956,11.022,399.024,166.926,50.201,159.189
C04914=1021.951,10.805,399.036,166.924,50.205,159.189
C04915=1021.945,10.589,399.049,166.921,50.209,159.190
C04916=1021.940,10.371,399.061,166.918,50.213,159.190
C04917=1021.935,10.154,399.074,166.917,50.217,159.191
C04918=1021.930,9.937,399.086,166.914,50.221,159.191
C04919=1021.924,9.688,399.100,166.911,50.226,159.191
C04920=1021.918,9.437,399.115,166.908,50.231,159.192
C04921=1021.912,9.188,399.129,166.906,50.235,159.192
C04922=1021.906,8.939,399.142,166.903,50.239,159.193
C04923=1021.899,8.689,399.157,166.900,50.244,159.193
C04924=1021.894,8.440,399.171,166.898,50.249,159.194
C04925=1021.888,8.191,399.186,166.895,50.253,159.194
C04926=1021.882,7.941,399.200,166.892,50.258,159.194
C04927=1021.877,7.691,399.214,166.890,50.263,159.195
C04928=1021.870,7.441,399.229,166.887,50.268,159.195
C04929=1021.865,7.192,399.243,166.884,50.272,159.196
C04930=1021.858,6.943,399.257,166.881,50.277,159.196
C04931=1021.852,6.693,399.271,166.879,50.281,159.196
C04932=1021.847,6.443,399.285,166.877,50.286,159.197
C04933=1021.841,6.194,399.299,166.873,50.291,159.197
C04934=1021.835,5.944,399.314,166.871,50.295,159.198
C04935=1021.829,5.695,399.328,166.868,50.300,159.198
C04936=1021.823,5.446,399.342,166.865,50.305,159.198
C04937=1021.817,5.196,399.356,166.862,50.309,159.199
C04938=1021.811,4.947,399.370,166.860,50.314,159.199
C04939=1021.805,4.697,399.384,166.857,50.319,159.200
C04940=1021.800,4.447,399.398,166.854,50.323,159.200
C04941=1021.794,4.198,399.413,166.852,50.328,159.201
C04942=1021.788,3.948,399.427,166.849,50.332,159.201
C04943=1021.783,3.699,399.441,166.846,50.337,159.201
C04944=1021.776,3.449,399.454,166.843,50.341,159.202
C04945=1021.770,3.200,399.469,166.841,50.346,159.202
C04946=1021.765,2.950,399.483,166.839,50.351,159.203
C04947=1021.759,2.701,399.497,166.835,50.355,159.203
C04948=1021.753,2.451,399.512,166.833,50.360,159.203
C04949=1021.747,2.201,399.525,166.830,50.364,159.204
C04950=1021.741,1.952,399.539,166.827,50.369,159.204
C04951=1021.735,1.703,399.553,166.824,50.373,159.204
C04952=1021.729,1.453,399.567,166.822,50.378,159.205
C04953=1021.724,1.203,399.581,166.819,50.382,159.205
C04954=1021.718,0.954,399.595,166.816,50.387,159.206
C04955=1021.713,0.704,399.609,166.814,50.392,159.206
C04956=1021.706,0.455,399.623,166.811,50.396,159.206
C04957=1021.700,0.205,399.637,166.809,50.401,159.207
C04958=1021.695,-0.044,399.651,166.805,50.405,159.207
C04959=1021.689,-0.294,399.665,166.803,50.410,159.208
C04960=1021.684,-0.543,399.679,166.800,50.414,159.208
C04961=1021.677,-0.793,399.694,166.797,50.419,159.208
C04962=1021.671,-1.042,399.707,166.794,50.423,159.209
C04963=1021.666,-1.292,399.721,166.792,50.427,159.209
C04964=1021.660,-1.542,399.735,166.789,50.432,159.209
C04965=1021.655,-1.791,399.749,166.786,50.436,159.210
C04966=1021.649,-2.041,399.763,166.784,50.441,159.210
C04967=1021.643,-2.290,399.777,166.781,50.445,159.211
C04968=1021.637,-2.540,399.791,166.779,50.450,159.211
C04969=1021.631,-2.789,399.805,166.775,50.455,159.211
C04970=1021.626,-3.039,399.818,166.773,50.459,159.212
C04971=1021.618,-3.387,399.838,166.769,50.466,159.212
C04972=1021.610,-3.735,399.857,166.765,50.472,159.213
C04973=1021.602,-4.083,399.877,166.761,50.478,159.213
C04974=1021.594,-4.430,399.896,166.757,50.485,159.214
C04975=1021.587,-4.712,399.911,166.754,50.490,159.214
C04976=1021.580,-4.993,399.926,166.752,50.495,159.215
C04977=1021.573,-5.273,399.942,166.749,50.500,159.215
C04978=1021.567,-5.555,399.957,166.745,50.505,159.215
C04979=1021.561,-5.805,399.970,166.742,50.510,159.216
C04980=1021.555,-6.054,399.984,166.740,50.515,159.216
C04981=1021.549,-6.304,399.998,166.737,50.519,159.217
C04982=1021.543,-6.553,400.011,166.734,50.524,159.217
C04983=1021.537,-6.803,400.025,166.732,50.529,159.218
C04984=1021.531,-7.052,400.038,166.729,50.533,159.218
C04985=1021.525,-7.302,400.051,166.726,50.538,159.218
C04986=1021.520,-7.552,400.065,166.723,50.542,159.219
C04987=1021.513,-7.801,400.078,166.720,50.547,159.219
C04988=1021.508,-8.051,400.092,166.717,50.552,159.220
C04989=1021.502,-8.300,400.105,166.715,50.556,159.220
C04990=1021.496,-8.549,400.119,166.712,50.561,159.220
C04991=1021.490,-8.799,400.132,166.709,50.565,159.221
C04992=1021.485,-9.049,400.145,166.707,50.570,159.221
C04993=1021.479,-9.298,400.159,166.703,50.575,159.221
C04994=1021.472,-9.548,400.173,166.701,50.579,159.222
C04995=1021.466,-9.798,400.186,166.699,50.584,159.222
C04996=1021.461,-10.048,400.199,166.695,50.589,159.222
C04997=1021.455,-10.297,400.213,166.693,50.593,159.223
C04998=1021.449,-10.546,400.226,166.690,50.598,159.223
C04999=1021.443,-10.796,400.240,166.687,50.603,159.224
C05000=1021.437,-11.045,400.253,166.684,50.607,159.224
C05001=1021.432,-11.295,400.266,166.682,50.612,159.224
C05002=1021.426,-11.545,400.279,166.678,50.616,159.225
C05003=1021.420,-11.794,400.293,166.676,50.621,159.225
C05004=1021.414,-12.044,400.306,166.673,50.625,159.225
C05005=1021.409,-12.294,400.320,166.670,50.630,159.226
C05006=1021.402,-12.543,400.333,166.667,50.634,159.226
C05007=1021.396,-12.792,400.346,166.665,50.639,159.227
C05008=1021.391,-13.042,400.359,166.662,50.643,159.227
C05009=1021.385,-13.292,400.373,166.659,50.648,159.227
C05010=1021.379,-13.541,400.387,166.657,50.652,159.228
C05011=1021.374,-13.791,400.399,166.653,50.657,159.228
C05012=1021.368,-14.041,400.413,166.651,50.662,159.228
C05013=1021.362,-14.290,400.426,166.648,50.666,159.229
C05014=1021.357,-14.540,400.439,166.645,50.671,159.229
C05015=1021.350,-14.790,400.453,166.642,50.675,159.229
C05016=1021.344,-15.039,400.466,166.640,50.680,159.230
C05017=1021.339,-15.289,400.479,166.636,50.684,159.230
C05018=1021.333,-15.538,400.492,166.634,50.688,159.230
C05019=1021.327,-15.788,400.506,166.632,50.693,159.231
C05020=1021.322,-16.037,400.518,166.628,50.698,159.231
C05021=1021.316,-16.286,400.532,166.626,50.702,159.232
C05022=1021.310,-16.536,400.544,166.623,50.707,159.232
C05023=1021.304,-16.786,400.558,166.620,50.712,159.232
C05024=1021.299,-17.036,400.571,166.618,50.717,159.233
C05025=1021.292,-17.285,400.584,166.614,50.721,159.233
C05026=1021.286,-17.535,400.596,166.612,50.726,159.234
C05027=1021.280,-17.784,400.610,166.609,50.730,159.234
C05028=1021.274,-18.034,400.622,166.606,50.735,159.234
C05029=1021.269,-18.284,400.635,166.604,50.740,159.235
C05030=1021.263,-18.533,400.649,166.600,50.744,159.235
C05031=1021.257,-18.783,400.661,166.598,50.749,159.235
C05032=1021.251,-19.032,400.675,166.595,50.753,159.236
C05033=1021.245,-19.282,400.687,166.592,50.758,159.236
C05034=1021.239,-19.531,400.700,166.589,50.763,159.236
C05035=1021.234,-19.781,400.713,166.586,50.768,159.237
C05036=1021.228,-20.031,400.726,166.583,50.772,159.237
C05037=1021.222,-20.280,400.739,166.581,50.777,159.238
C05038=1021.216,-20.530,400.752,166.577,50.781,159.238
C05039=1021.210,-20.810,400.766,166.574,50.786,159.238
C05040=1021.203,-21.089,400.780,166.571,50.791,159.239
C05041=1021.197,-21.368,400.795,166.568,50.797,159.239
C05042=1021.190,-21.648,400.809,166.565,50.801,159.239
C05043=1021.184,-21.897,400.822,166.562,50.807,159.240
C05044=1021.179,-22.146,400.835,166.560,50.811,159.240
C05045=1021.173,-22.396,400.847,166.556,50.816,159.241
C05046=1021.167,-22.645,400.860,166.554,50.820,159.241
C05047=1021.161,-22.895,400.874,166.551,50.825,159.241
C05048=1021.155,-23.145,400.886,166.548,50.829,159.242
C05049=1021.149,-23.395,400.899,166.545,50.833,159.242
C05050=1021.144,-23.644,400.912,166.542,50.839,159.242
C05051=1021.138,-23.894,400.924,166.539,50.843,159.243
C05052=1021.132,-24.144,400.937,166.537,50.848,159.243
C05053=1021.126,-24.393,400.950,166.533,50.852,159.243
C05054=1021.121,-24.642,400.963,166.531,50.857,159.244
C05055=1021.115,-24.892,400.975,166.529,50.861,159.244
C05056=1021.110,-25.142,400.988,166.525,50.865,159.244
C05057=1021.103,-25.391,401.001,166.523,50.870,159.245
C05058=1021.097,-25.641,401.014,166.520,50.874,159.245
C05059=1021.092,-25.890,401.026,166.517,50.880,159.245
C05060=1021.086,-26.140,401.038,166.514,50.884,159.246
C05061=1021.080,-26.390,401.052,166.511,50.888,159.246
C05062=1021.075,-26.640,401.065,166.508,50.893,159.246
C05063=1021.070,-26.889,401.077,166.506,50.897,159.247
C05064=1021.064,-27.139,401.090,166.502,50.902,159.247
C05065=1021.058,-27.389,401.102,166.500,50.907,159.247
C05066=1021.052,-27.639,401.115,166.497,50.911,159.248
C05067=1021.046,-27.888,401.127,166.494,50.916,159.248
C05068=1021.040,-28.137,401.140,166.492,50.920,159.248
C05069=1021.034,-28.387,401.153,166.488,50.925,159.249
C05070=1021.028,-28.637,401.165,166.486,50.929,159.249
C05071=1021.023,-28.886,401.177,166.482,50.934,159.249
C05072=1021.016,-29.136,401.189,166.480,50.939,159.250
C05073=1021.011,-29.385,401.202,166.477,50.944,159.250
C05074=1021.005,-29.635,401.214,166.474,50.948,159.250
C05075=1020.999,-29.884,401.227,166.472,50.953,159.251
C05076=1020.993,-30.134,401.239,166.468,50.957,159.251
C05077=1020.988,-30.384,401.252,166.466,50.962,159.252
C05078=1020.982,-30.633,401.264,166.462,50.967,159.252
C05079=1020.976,-30.883,401.276,166.460,50.971,159.252
C05080=1020.970,-31.133,401.289,166.456,50.976,159.252
C05081=1020.964,-31.382,401.301,166.454,50.981,159.253
C05082=1020.958,-31.632,401.313,166.451,50.985,159.253
C05083=1020.953,-31.882,401.325,166.448,50.989,159.253
C05084=1020.948,-32.132,401.337,166.446,50.994,159.254
C05085=1020.942,-32.382,401.350,166.442,50.999,159.254
C05086=1020.936,-32.630,401.361,166.440,51.004,159.255
C05087=1020.930,-32.880,401.374,166.436,51.008,159.255
C05088=1020.924,-33.130,401.387,166.434,51.013,159.255
C05089=1020.918,-33.379,401.399,166.430,51.017,159.255
C05090=1020.913,-33.629,401.411,166.428,51.022,159.256
C05091=1020.907,-33.879,401.424,166.426,51.026,159.256
C05092=1020.901,-34.128,401.435,166.422,51.031,159.256
C05093=1020.895,-34.378,401.448,166.420,51.036,159.257
C05094=1020.890,-34.628,401.459,166.416,51.040,159.257
C05095=1020.884,-34.878,401.472,166.414,51.044,159.257
C05096=1020.878,-35.127,401.485,166.410,51.050,159.258
C05097=1020.873,-35.377,401.497,166.408,51.054,159.258
C05098=1020.866,-35.626,401.509,166.405,51.058,159.258
C05099=1020.861,-35.875,401.521,166.402,51.063,159.259
C05100=1020.855,-36.126,401.533,166.399,51.067,159.259
C05101=1020.850,-36.375,401.545,166.396,51.072,159.259
C05102=1020.844,-36.625,401.557,166.394,51.077,159.260
C05103=1020.837,-36.903,401.571,166.390,51.082,159.260
C05104=1020.831,-37.182,401.584,166.387,51.087,159.260
C05105=1020.825,-37.460,401.598,166.383,51.091,159.261
C05106=1020.818,-37.739,401.612,166.380,51.097,159.261
C05107=1020.813,-37.988,401.623,166.378,51.101,159.261
C05108=1020.807,-38.238,401.636,166.375,51.106,159.262
C05109=1020.801,-38.487,401.647,166.372,51.110,159.262
C05110=1020.795,-38.737,401.660,166.369,51.114,159.262
C05111=1020.790,-38.987,401.672,166.366,51.120,159.263
C05112=1020.784,-39.237,401.684,166.363,51.124,159.263
C05113=1020.778,-39.487,401.697,166.360,51.128,159.263
C05114=1020.773,-39.736,401.707,166.358,51.133,159.264
C05115=1020.767,-39.986,401.720,166.354,51.138,159.264
C05116=1020.761,-40.235,401.731,166.352,51.142,159.264
C05117=1020.755,-40.485,401.743,166.348,51.147,159.264
C05118=1020.749,-40.734,401.755,166.346,51.152,159.265
C05119=1020.744,-40.984,401.767,166.343,51.156,159.265
C05120=1020.738,-41.234,401.779,166.340,51.161,159.266
C05121=1020.732,-41.483,401.790,166.337,51.165,159.266
C05122=1020.727,-41.733,401.803,166.334,51.170,159.266
C05123=1020.721,-41.983,401.813,166.332,51.175,159.267
C05124=1020.715,-42.233,401.826,166.328,51.179,159.267
C05125=1020.709,-42.482,401.837,166.326,51.184,159.267
C05126=1020.703,-42.732,401.849,166.322,51.189,159.267
C05127=1020.698,-42.982,401.860,166.320,51.193,159.268
C05128=1020.692,-43.231,401.873,166.316,51.198,159.268
C05129=1020.687,-43.481,401.884,166.314,51.202,159.268
C05130=1020.681,-43.730,401.896,166.311,51.207,159.269
C05131=1020.675,-43.981,401.908,166.308,51.211,159.269
C05132=1020.669,-44.229,401.919,166.304,51.216,159.269
C05133=1020.663,-44.480,401.931,166.302,51.221,159.270
C05134=1020.657,-44.729,401.943,166.299,51.225,159.270
C05135=1020.652,-44.979,401.955,166.296,51.230,159.270
C05136=1020.646,-45.228,401.966,166.293,51.235,159.271
C05137=1020.641,-45.478,401.978,166.290,51.239,159.271
C05138=1020.634,-45.728,401.990,166.288,51.243,159.271
C05139=1020.629,-45.977,402.001,166.284,51.248,159.271
C05140=1020.624,-46.227,402.013,166.282,51.252,159.272
C05141=1020.617,-46.477,402.025,166.278,51.257,159.272
C05142=1020.612,-46.727,402.036,166.276,51.262,159.272
C05143=1020.606,-46.975,402.048,166.272,51.266,159.273
C05144=1020.601,-47.226,402.059,166.270,51.271,159.273
C05145=1020.595,-47.475,402.070,166.267,51.276,159.273
C05146=1020.589,-47.725,402.083,166.264,51.280,159.274
C05147=1020.583,-47.975,402.094,166.260,51.284,159.274
C05148=1020.578,-48.225,402.105,166.258,51.289,159.274
C05149=1020.572,-48.473,402.117,166.256,51.294,159.275
C05150=1020.567,-48.724,402.129,166.252,51.298,159.275
C05151=1020.561,-48.973,402.140,166.249,51.302,159.275
C05152=1020.556,-49.223,402.152,166.246,51.307,159.275
C05153=1020.550,-49.473,402.164,166.244,51.312,159.276
C05154=1020.544,-49.723,402.174,166.240,51.316,159.276
C05155=1020.539,-49.972,402.187,166.237,51.320,159.276
C05156=1020.533,-50.222,402.198,166.234,51.326,159.276
C05157=1020.528,-50.472,402.209,166.232,51.330,159.277
C05158=1020.522,-50.721,402.221,166.229,51.334,159.277
C05159=1020.517,-50.970,402.232,166.225,51.338,159.277
C05160=1020.510,-51.221,402.244,166.223,51.343,159.278
C05161=1020.504,-51.470,402.254,166.220,51.348,159.278
C05162=1020.499,-51.720,402.265,166.216,51.353,159.278
C05163=1020.492,-51.970,402.277,166.214,51.357,159.278
C05164=1020.487,-52.219,402.287,166.211,51.362,159.279
C05165=1020.481,-52.469,402.298,166.208,51.367,159.279
C05166=1020.476,-52.719,402.310,166.205,51.372,159.280
C05167=1020.469,-52.997,402.322,166.202,51.377,159.280
C05168=1020.463,-53.276,402.335,166.198,51.382,159.280
C05169=1020.456,-53.555,402.347,166.195,51.388,159.281
C05170=1020.449,-53.834,402.360,166.192,51.393,159.281
C05171=1020.444,-54.083,402.370,166.188,51.397,159.281
C05172=1020.438,-54.333,402.381,166.186,51.402,159.282
C05173=1020.432,-54.582,402.392,166.183,51.407,159.282
C05174=1020.426,-54.833,402.404,166.179,51.412,159.282
C05175=1020.421,-55.082,402.415,166.177,51.416,159.282
C05176=1020.415,-55.332,402.426,166.173,51.421,159.283
C05177=1020.409,-55.581,402.437,166.171,51.426,159.283
C05178=1020.403,-55.831,402.448,166.167,51.430,159.283
C05179=1020.397,-56.081,402.459,166.165,51.435,159.284
C05180=1020.391,-56.330,402.470,166.162,51.440,159.284
C05181=1020.386,-56.580,402.481,166.159,51.444,159.284
C05182=1020.380,-56.829,402.491,166.156,51.449,159.285
C05183=1020.375,-57.080,402.502,166.152,51.454,159.285
C05184=1020.369,-57.329,402.513,166.150,51.458,159.285
C05185=1020.363,-57.580,402.524,166.146,51.463,159.285
C05186=1020.357,-57.829,402.535,166.144,51.467,159.286
C05187=1020.352,-58.079,402.546,166.141,51.472,159.286
C05188=1020.346,-58.328,402.557,166.138,51.477,159.286
C05189=1020.340,-58.577,402.568,166.135,51.481,159.286
C05190=1020.334,-58.827,402.579,166.132,51.486,159.287
C05191=1020.329,-59.077,402.590,166.129,51.491,159.287
C05192=1020.323,-59.328,402.601,166.127,51.496,159.288
C05193=1020.318,-59.577,402.612,166.123,51.500,159.288
C05194=1020.312,-59.827,402.622,166.119,51.505,159.288
C05195=1020.306,-60.076,402.633,166.117,51.509,159.288
C05196=1020.300,-60.326,402.644,166.114,51.514,159.289
C05197=1020.295,-60.575,402.655,166.111,51.518,159.289
C05198=1020.289,-60.825,402.665,166.107,51.523,159.289
C05199=1020.284,-61.075,402.676,166.105,51.528,159.289
C05200=1020.278,-61.324,402.687,166.102,51.532,159.290
C05201=1020.273,-61.574,402.698,166.099,51.536,159.290
C05202=1020.267,-61.823,402.709,166.096,51.542,159.290
C05203=1020.262,-62.074,402.720,166.093,51.546,159.291
C05204=1020.256,-62.323,402.730,166.090,51.550,159.291
C05205=1020.250,-62.573,402.741,166.087,51.555,159.291
C05206=1020.244,-62.823,402.753,166.084,51.560,159.291
C05207=1020.238,-63.073,402.763,166.081,51.564,159.292
C05208=1020.233,-63.322,402.774,166.078,51.569,159.292
C05209=1020.227,-63.572,402.784,166.076,51.574,159.292
C05210=1020.221,-63.822,402.795,166.072,51.578,159.292
C05211=1020.216,-64.071,402.805,166.069,51.582,159.293
C05212=1020.211,-64.321,402.817,166.066,51.587,159.293
C05213=1020.205,-64.571,402.828,166.063,51.591,159.293
C05214=1020.200,-64.821,402.838,166.060,51.596,159.293
C05215=1020.194,-65.070,402.849,166.058,51.601,159.294
C05216=1020.188,-65.320,402.860,166.054,51.605,159.294
C05217=1020.183,-65.570,402.870,166.051,51.609,159.294
C05218=1020.177,-65.819,402.880,166.048,51.615,159.295
C05219=1020.172,-66.068,402.891,166.046,51.619,159.295
C05220=1020.166,-66.318,402.901,166.042,51.623,159.295
C05221=1020.161,-66.568,402.912,166.040,51.627,159.295
C05222=1020.155,-66.818,402.922,166.036,51.632,159.295
C05223=1020.149,-67.067,402.933,166.033,51.636,159.296
C05224=1020.144,-67.317,402.945,166.030,51.642,159.296
C05225=1020.139,-67.567,402.955,166.028,51.646,159.296
C05226=1020.133,-67.817,402.966,166.024,51.650,159.296
C05227=1020.128,-68.067,402.976,166.021,51.654,159.297
C05228=1020.122,-68.316,402.987,166.018,51.659,159.297
C05229=1020.116,-68.566,402.998,166.015,51.663,159.297
C05230=1020.111,-68.816,403.008,166.012,51.669,159.298
C05231=1020.105,-69.096,403.020,166.009,51.673,159.298
C05232=1020.099,-69.376,403.031,166.005,51.678,159.298
C05233=1020.093,-69.655,403.043,166.002,51.683,159.298
C05234=1020.086,-69.935,403.055,165.999,51.688,159.299
C05235=1020.080,-70.185,403.065,165.996,51.692,159.299
C05236=1020.076,-70.435,403.076,165.992,51.697,159.299
C05237=1020.071,-70.685,403.087,165.990,51.701,159.299
C05238=1020.065,-70.934,403.097,165.987,51.705,159.300
C05239=1020.059,-71.184,403.108,165.984,51.711,159.300
C05240=1020.054,-71.434,403.118,165.982,51.715,159.300
C05241=1020.048,-71.684,403.129,165.978,51.719,159.300
C05242=1020.043,-71.933,403.139,165.975,51.724,159.301
C05243=1020.038,-72.183,403.149,165.972,51.728,159.301
C05244=1020.032,-72.432,403.160,165.969,51.732,159.301
C05245=1020.027,-72.682,403.170,165.966,51.737,159.301
C05246=1020.021,-72.932,403.181,165.963,51.741,159.301
C05247=1020.016,-73.181,403.191,165.961,51.745,159.302
C05248=1020.011,-73.431,403.201,165.957,51.750,159.302
C05249=1020.005,-73.681,403.212,165.954,51.754,159.302
C05250=1019.999,-73.931,403.222,165.951,51.759,159.302
C05251=1019.994,-74.180,403.233,165.948,51.763,159.303
C05252=1019.989,-74.430,403.243,165.945,51.768,159.303
C05253=1019.983,-74.680,403.253,165.942,51.772,159.303
C05254=1019.978,-74.930,403.263,165.939,51.777,159.303
C05255=1019.972,-75.180,403.274,165.936,51.781,159.304
C05256=1019.966,-75.429,403.284,165.933,51.786,159.304
C05257=1019.961,-75.679,403.293,165.930,51.790,159.304
C05258=1019.956,-75.929,403.304,165.927,51.795,159.304
C05259=1019.950,-76.179,403.314,165.925,51.800,159.305
C05260=1019.944,-76.428,403.324,165.921,51.804,159.305
C05261=1019.939,-76.678,403.334,165.917,51.809,159.305
C05262=1019.934,-76.928,403.344,165.915,51.813,159.305
C05263=1019.928,-77.178,403.354,165.912,51.818,159.306
C05264=1019.922,-77.428,403.364,165.909,51.823,159.306
C05265=1019.917,-77.676,403.374,165.905,51.827,159.306
C05266=1019.911,-77.927,403.384,165.903,51.831,159.306
C05267=1019.906,-78.177,403.395,165.899,51.836,159.306
C05268=1019.900,-78.426,403.404,165.897,51.840,159.307
C05269=1019.895,-78.676,403.414,165.894,51.845,159.307
C05270=1019.890,-78.926,403.424,165.891,51.850,159.307
C05271=1019.885,-79.175,403.434,165.887,51.854,159.307
C05272=1019.879,-79.425,403.443,165.885,51.858,159.308
C05273=1019.873,-79.675,403.454,165.881,51.863,159.308
C05274=1019.868,-79.924,403.464,165.879,51.867,159.308
C05275=1019.863,-80.174,403.474,165.875,51.872,159.308
C05276=1019.856,-80.424,403.484,165.873,51.877,159.309
C05277=1019.852,-80.673,403.494,165.870,51.881,159.309
C05278=1019.845,-80.923,403.503,165.866,51.886,159.309
C05279=1019.840,-81.174,403.513,165.864,51.891,159.310
C05280=1019.835,-81.423,403.522,165.860,51.895,159.310
C05281=1019.829,-81.673,403.532,165.858,51.900,159.310
C05282=1019.823,-81.923,403.542,165.854,51.905,159.310
C05283=1019.817,-82.172,403.551,165.851,51.910,159.310
C05284=1019.812,-82.422,403.561,165.848,51.914,159.311
C05285=1019.806,-82.672,403.570,165.845,51.918,159.311
C05286=1019.801,-82.921,403.580,165.843,51.923,159.311
C05287=1019.795,-83.171,403.590,165.839,51.928,159.311
C05288=1019.790,-83.421,403.600,165.835,51.933,159.312
C05289=1019.784,-83.671,403.609,165.833,51.938,159.312
C05290=1019.779,-83.921,403.619,165.830,51.942,159.312
C05291=1019.773,-84.170,403.628,165.827,51.946,159.312
C05292=1019.768,-84.420,403.638,165.824,51.951,159.313
C05293=1019.762,-84.669,403.647,165.821,51.955,159.313
C05294=1019.757,-84.919,403.657,165.818,51.960,159.313
C05295=1019.750,-85.201,403.667,165.815,51.966,159.314
C05296=1019.744,-85.484,403.678,165.811,51.970,159.314
C05297=1019.738,-85.765,403.689,165.807,51.976,159.314
C05298=1019.732,-86.047,403.700,165.804,51.981,159.314
C05299=1019.726,-86.297,403.709,165.801,51.986,159.315
C05300=1019.721,-86.547,403.719,165.798,51.990,159.315
C05301=1019.715,-86.796,403.728,165.795,51.994,159.315
C05302=1019.710,-87.046,403.738,165.792,52.000,159.315
C05303=1019.704,-87.296,403.747,165.789,52.004,159.316
C05304=1019.699,-87.546,403.757,165.786,52.009,159.316
C05305=1019.693,-87.795,403.766,165.782,52.013,159.316
C05306=1019.688,-88.045,403.775,165.780,52.017,159.316
C05307=1019.683,-88.295,403.785,165.776,52.022,159.316
C05308=1019.677,-88.544,403.794,165.774,52.027,159.317
C05309=1019.672,-88.794,403.804,165.771,52.032,159.317
C05310=1019.666,-89.044,403.813,165.768,52.036,159.317
C05311=1019.661,-89.294,403.823,165.764,52.040,159.317
C05312=1019.655,-89.543,403.832,165.762,52.045,159.317
C05313=1019.650,-89.794,403.842,165.758,52.049,159.318
C05314=1019.645,-90.043,403.851,165.756,52.054,159.318
C05315=1019.638,-90.293,403.861,165.753,52.059,159.318
C05316=1019.634,-90.543,403.870,165.749,52.063,159.318
C05317=1019.628,-90.792,403.879,165.746,52.068,159.319
C05318=1019.623,-91.043,403.888,165.743,52.072,159.319
C05319=1019.618,-91.292,403.897,165.740,52.077,159.319
C05320=1019.612,-91.542,403.908,165.737,52.081,159.319
C05321=1019.607,-91.792,403.916,165.734,52.085,159.319
C05322=1019.601,-92.042,403.926,165.731,52.090,159.320
C05323=1019.596,-92.292,403.935,165.728,52.094,159.320
C05324=1019.591,-92.541,403.944,165.725,52.100,159.320
C05325=1019.585,-92.791,403.954,165.722,52.104,159.320
C05326=1019.580,-93.040,403.963,165.719,52.108,159.321
C05327=1019.575,-93.290,403.972,165.716,52.113,159.321
C05328=1019.569,-93.540,403.981,165.713,52.117,159.321
C05329=1019.564,-93.789,403.990,165.710,52.122,159.321
C05330=1019.559,-94.040,404.000,165.707,52.126,159.321
C05331=1019.553,-94.289,404.009,165.704,52.130,159.322
C05332=1019.548,-94.539,404.018,165.701,52.135,159.322
C05333=1019.542,-94.789,404.028,165.698,52.139,159.322
C05334=1019.537,-95.039,404.036,165.695,52.144,159.322
C05335=1019.532,-95.288,404.046,165.692,52.148,159.322
C05336=1019.526,-95.539,404.055,165.688,52.153,159.322
C05337=1019.521,-95.788,404.065,165.686,52.157,159.323
C05338=1019.516,-96.038,404.073,165.682,52.162,159.323
C05339=1019.511,-96.287,404.082,165.680,52.166,159.323
C05340=1019.505,-96.538,404.092,165.676,52.171,159.323
C05341=1019.500,-96.787,404.101,165.674,52.175,159.324
C05342=1019.495,-97.037,404.110,165.670,52.179,159.324
C05343=1019.490,-97.287,404.119,165.668,52.184,159.324
C05344=1019.485,-97.536,404.129,165.665,52.188,159.324
C05345=1019.479,-97.786,404.137,165.662,52.193,159.324
C05346=1019.473,-98.036,404.147,165.659,52.197,159.325
C05347=1019.468,-98.286,404.155,165.655,52.201,159.325
C05348=1019.463,-98.535,404.164,165.652,52.207,159.325
C05349=1019.458,-98.785,404.173,165.650,52.211,159.325
C05350=1019.452,-99.035,404.182,165.646,52.216,159.325
C05351=1019.447,-99.285,404.191,165.644,52.220,159.326
C05352=1019.442,-99.535,404.199,165.640,52.225,159.326
C05353=1019.436,-99.784,404.208,165.638,52.229,159.326
C05354=1019.430,-100.034,404.217,165.634,52.233,159.326
C05355=1019.425,-100.284,404.226,165.631,52.239,159.327
C05356=1019.420,-100.534,404.235,165.628,52.243,159.327
C05357=1019.415,-100.784,404.243,165.625,52.248,159.327
C05358=1019.409,-101.034,404.252,165.622,52.252,159.327
C05359=1019.403,-101.318,404.262,165.619,52.257,159.328
C05360=1019.397,-101.601,404.272,165.614,52.262,159.327
C05361=1019.391,-101.885,404.282,165.611,52.268,159.328
C05362=1019.385,-102.170,404.292,165.608,52.273,159.328
C05363=1019.379,-102.419,404.301,165.606,52.277,159.328
C05364=1019.374,-102.669,404.310,165.602,52.282,159.329
C05365=1019.369,-102.919,404.319,165.600,52.286,159.329
C05366=1019.364,-103.169,404.327,165.596,52.291,159.329
C05367=1019.359,-103.419,404.336,165.593,52.295,159.329
C05368=1019.353,-103.668,404.344,165.590,52.300,159.329
C05369=1019.347,-103.919,404.353,165.586,52.304,159.329
C05370=1019.342,-104.168,404.361,165.584,52.309,159.330
C05371=1019.337,-104.418,404.370,165.580,52.313,159.330
C05372=1019.331,-104.667,404.379,165.578,52.317,159.330
C05373=1019.326,-104.917,404.388,165.575,52.323,159.330
C05374=1019.321,-105.167,404.396,165.572,52.327,159.331
C05375=1019.316,-105.417,404.405,165.569,52.332,159.331
C05376=1019.311,-105.666,404.414,165.566,52.336,159.331
C05377=1019.306,-105.916,404.422,165.562,52.341,159.331
C05378=1019.300,-106.166,404.431,165.560,52.345,159.331
C05379=1019.295,-106.416,404.440,165.556,52.350,159.332
C05380=1019.289,-106.666,404.448,165.554,52.354,159.332
C05381=1019.284,-106.916,404.456,165.550,52.358,159.332
C05382=1019.279,-107.165,404.465,165.548,52.363,159.332
C05383=1019.274,-107.415,404.473,165.544,52.367,159.332
C05384=1019.268,-107.665,404.482,165.542,52.372,159.333
C05385=1019.263,-107.914,404.490,165.538,52.376,159.333
C05386=1019.258,-108.165,404.498,165.536,52.381,159.333
C05387=1019.253,-108.415,404.507,165.532,52.385,159.333
C05388=1019.248,-108.664,404.515,165.530,52.390,159.333
C05389=1019.242,-108.914,404.524,165.526,52.395,159.334
C05390=1019.237,-109.164,404.532,165.523,52.400,159.334
C05391=1019.231,-109.413,404.540,165.520,52.404,159.334
C05392=1019.226,-109.663,404.549,165.517,52.408,159.334
C05393=1019.221,-109.913,404.556,165.514,52.413,159.334
C05394=1019.215,-110.163,404.565,165.511,52.417,159.334
C05395=1019.210,-110.413,404.573,165.508,52.422,159.335
C05396=1019.205,-110.662,404.582,165.505,52.426,159.335
C05397=1019.200,-110.912,404.590,165.502,52.431,159.335
C05398=1019.195,-111.162,404.598,165.499,52.436,159.335
C05399=1019.189,-111.412,404.606,165.497,52.440,159.336
///RCONF 1,0,0,0,1,0,0,0,0,0,0,0,0,0,0,0,0,0,0,0,0,0,0,0
C05400=1019.184,-111.662,404.615,165.493,52.445,159.336
C05401=1019.178,-111.911,404.623,165.490,52.449,159.336
C05402=1019.173,-112.161,404.631,165.487,52.454,159.336
C05403=1019.168,-112.411,404.639,165.484,52.458,159.336
C05404=1019.163,-112.661,404.648,165.481,52.463,159.336
C05405=1019.157,-112.911,404.656,165.478,52.467,159.337
C05406=1019.152,-113.160,404.665,165.475,52.472,159.337
C05407=1019.147,-113.411,404.672,165.472,52.476,159.337
C05408=1019.142,-113.660,404.681,165.469,52.481,159.337
C05409=1019.137,-113.910,404.689,165.466,52.485,159.337
C05410=1019.131,-114.160,404.696,165.463,52.490,159.338
C05411=1019.126,-114.410,404.705,165.460,52.494,159.338
C05412=1019.120,-114.660,404.713,165.457,52.499,159.338
C05413=1019.116,-114.910,404.721,165.453,52.503,159.338
C05414=1019.111,-115.159,404.729,165.451,52.508,159.339
C05415=1019.106,-115.409,404.738,165.447,52.513,159.339
C05416=1019.100,-115.659,404.745,165.445,52.517,159.339
C05417=1019.095,-115.908,404.753,165.441,52.522,159.339
C05418=1019.090,-116.159,404.761,165.439,52.526,159.339
C05419=1019.084,-116.408,404.770,165.435,52.531,159.339
C05420=1019.078,-116.658,404.778,165.433,52.535,159.340
C05421=1019.073,-116.908,404.785,165.429,52.540,159.340
C05422=1019.069,-117.157,404.794,165.427,52.544,159.340
C05423=1019.063,-117.441,404.803,165.424,52.549,159.340
C05424=1019.057,-117.725,404.811,165.419,52.555,159.340
C05425=1019.051,-118.009,404.820,165.416,52.560,159.341
C05426=1019.045,-118.294,404.830,165.413,52.565,159.341
C05427=1019.040,-118.544,404.837,165.410,52.569,159.341
C05428=1019.034,-118.793,404.845,165.407,52.574,159.341
C05429=1019.030,-119.044,404.853,165.403,52.579,159.341
C05430=1019.024,-119.293,404.861,165.401,52.583,159.342
C05431=1019.019,-119.543,404.868,165.397,52.588,159.342
C05432=1019.014,-119.792,404.877,165.395,52.592,159.342
C05433=1019.008,-120.042,404.884,165.391,52.597,159.342
C05434=1019.003,-120.292,404.892,165.389,52.602,159.343
C05435=1018.998,-120.542,404.900,165.385,52.606,159.343
C05436=1018.994,-120.792,404.908,165.383,52.611,159.343
C05437=1018.988,-121.041,404.916,165.379,52.615,159.343
C05438=1018.983,-121.292,404.923,165.377,52.620,159.343
C05439=1018.977,-121.542,404.932,165.373,52.624,159.343
C05440=1018.972,-121.791,404.939,165.371,52.629,159.344
C05441=1018.967,-122.041,404.946,165.367,52.633,159.344
C05442=1018.962,-122.291,404.955,165.365,52.638,159.344
C05443=1018.956,-122.541,404.962,165.361,52.642,159.344
C05444=1018.952,-122.791,404.969,165.359,52.647,159.344
C05445=1018.947,-123.040,404.978,165.355,52.651,159.344
C05446=1018.941,-123.290,404.985,165.353,52.656,159.345
C05447=1018.936,-123.541,404.993,165.350,52.661,159.345
C05448=1018.931,-123.789,405.000,165.347,52.665,159.345
C05449=1018.926,-124.040,405.008,165.344,52.670,159.345
C05450=1018.921,-124.290,405.016,165.341,52.674,159.346
C05451=1018.915,-124.539,405.023,165.338,52.679,159.346
C05452=1018.910,-124.789,405.031,165.335,52.683,159.346
C05453=1018.905,-125.039,405.039,165.331,52.688,159.346
C05454=1018.900,-125.289,405.046,165.329,52.692,159.346
C05455=1018.895,-125.539,405.054,165.325,52.697,159.346
C05456=1018.889,-125.788,405.061,165.322,52.702,159.346
C05457=1018.885,-126.038,405.069,165.320,52.707,159.347
C05458=1018.879,-126.288,405.076,165.316,52.711,159.347
C05459=1018.874,-126.538,405.084,165.314,52.716,159.347
